C01801=1111.300,173.599,-64.329,-179.246,9.058,149.558
C01802=1111.305,173.385,-64.308,-179.248,9.055,149.558
C01803=1111.309,173.172,-64.289,-179.250,9.053,149.558
C01804=1111.313,172.959,-64.268,-179.252,9.051,149.558
C01805=1111.317,172.746,-64.249,-179.254,9.048,149.558
C01806=1111.321,172.532,-64.228,-179.255,9.045,149.557
C01807=1111.325,172.283,-64.204,-179.258,9.042,149.557
C01808=1111.329,172.035,-64.181,-179.260,9.039,149.557
C01809=1111.334,171.786,-64.158,-179.261,9.037,149.557
C01810=1111.339,171.536,-64.135,-179.264,9.033,149.557
C01811=1111.343,171.288,-64.111,-179.267,9.030,149.557
C01812=1111.348,171.039,-64.087,-179.268,9.028,149.557
C01813=1111.353,170.790,-64.064,-179.271,9.025,149.557
C01814=1111.357,170.541,-64.040,-179.273,9.021,149.557
C01815=1111.362,170.292,-64.017,-179.275,9.018,149.556
C01816=1111.366,170.043,-63.994,-179.277,9.016,149.556
C01817=1111.370,169.795,-63.970,-179.280,9.012,149.556
C01818=1111.375,169.546,-63.947,-179.282,9.009,149.556
C01819=1111.380,169.297,-63.924,-179.284,9.007,149.556
C01820=1111.384,169.048,-63.900,-179.286,9.004,149.556
C01821=1111.389,168.799,-63.877,-179.288,9.000,149.556
C01822=1111.393,168.550,-63.854,-179.290,8.998,149.556
C01823=1111.398,168.301,-63.831,-179.292,8.994,149.555
C01824=1111.403,168.053,-63.808,-179.295,8.991,149.555
C01825=1111.408,167.804,-63.784,-179.297,8.988,149.555
C01826=1111.412,167.555,-63.762,-179.299,8.985,149.555
C01827=1111.416,167.306,-63.738,-179.301,8.982,149.555
C01828=1111.421,167.057,-63.715,-179.304,8.979,149.555
C01829=1111.426,166.808,-63.692,-179.305,8.976,149.555
C01830=1111.430,166.559,-63.669,-179.308,8.973,149.555
C01831=1111.435,166.310,-63.645,-179.310,8.970,149.555
C01832=1111.439,166.061,-63.622,-179.312,8.967,149.555
C01833=1111.445,165.813,-63.599,-179.314,8.964,149.554
C01834=1111.449,165.564,-63.576,-179.316,8.961,149.554
C01835=1111.453,165.315,-63.553,-179.319,8.958,149.554
C01836=1111.458,165.066,-63.530,-179.321,8.954,149.554
C01837=1111.462,164.817,-63.507,-179.323,8.952,149.554
C01838=1111.467,164.568,-63.483,-179.325,8.949,149.554
C01839=1111.472,164.318,-63.461,-179.327,8.945,149.554
C01840=1111.476,164.070,-63.438,-179.330,8.942,149.554
C01841=1111.481,163.821,-63.415,-179.331,8.940,149.553
C01842=1111.486,163.572,-63.392,-179.334,8.936,149.553
C01843=1111.489,163.324,-63.369,-179.336,8.933,149.553
C01844=1111.494,163.075,-63.346,-179.338,8.930,149.553
C01845=1111.498,162.825,-63.324,-179.340,8.927,149.553
C01846=1111.504,162.577,-63.301,-179.342,8.924,149.553
C01847=1111.508,162.328,-63.277,-179.344,8.921,149.553
C01848=1111.512,162.079,-63.254,-179.347,8.917,149.553
C01849=1111.517,161.829,-63.232,-179.349,8.914,149.552
C01850=1111.521,161.581,-63.209,-179.351,8.912,149.552
C01851=1111.527,161.332,-63.186,-179.353,8.908,149.552
C01852=1111.531,161.084,-63.163,-179.356,8.905,149.552
C01853=1111.536,160.834,-63.141,-179.358,8.902,149.552
C01854=1111.540,160.585,-63.117,-179.360,8.898,149.552
C01855=1111.544,160.373,-63.098,-179.362,8.896,149.551
C01856=1111.548,160.159,-63.079,-179.364,8.893,149.551
C01857=1111.552,159.945,-63.059,-179.365,8.891,149.551
C01858=1111.556,159.731,-63.040,-179.368,8.888,149.551
C01859=1111.560,159.518,-63.020,-179.369,8.885,149.551
C01860=1111.564,159.305,-63.000,-179.371,8.883,149.551
C01861=1111.568,159.091,-62.981,-179.373,8.879,149.551
C01862=1111.572,158.877,-62.962,-179.375,8.877,149.551
C01863=1111.576,158.629,-62.939,-179.377,8.873,149.550
C01864=1111.581,158.379,-62.917,-179.379,8.871,149.550
C01865=1111.585,158.131,-62.894,-179.381,8.867,149.550
C01866=1111.590,157.882,-62.871,-179.383,8.864,149.550
C01867=1111.595,157.633,-62.849,-179.385,8.861,149.550
C01868=1111.599,157.384,-62.826,-179.388,8.857,149.550
C01869=1111.604,157.135,-62.804,-179.390,8.854,149.550
C01870=1111.608,156.887,-62.781,-179.392,8.851,149.549
C01871=1111.613,156.637,-62.758,-179.394,8.848,149.549
C01872=1111.617,156.388,-62.736,-179.396,8.845,149.549
C01873=1111.623,156.139,-62.713,-179.398,8.841,149.549
C01874=1111.627,155.891,-62.690,-179.400,8.838,149.549
C01875=1111.631,155.641,-62.668,-179.403,8.835,149.549
C01876=1111.637,155.392,-62.646,-179.405,8.831,149.548
C01877=1111.641,155.144,-62.623,-179.407,8.828,149.548
C01878=1111.645,154.894,-62.601,-179.409,8.824,149.548
C01879=1111.650,154.646,-62.578,-179.412,8.821,149.548
C01880=1111.654,154.397,-62.556,-179.414,8.818,149.548
C01881=1111.659,154.148,-62.535,-179.415,8.815,149.547
C01882=1111.664,153.899,-62.511,-179.417,8.812,149.547
C01883=1111.668,153.650,-62.489,-179.420,8.808,149.547
C01884=1111.673,153.401,-62.467,-179.422,8.805,149.547
C01885=1111.678,153.152,-62.444,-179.424,8.801,149.547
C01886=1111.682,152.902,-62.422,-179.426,8.798,149.546
C01887=1111.687,152.654,-62.400,-179.428,8.794,149.546
C01888=1111.692,152.405,-62.377,-179.430,8.791,149.546
C01889=1111.697,152.156,-62.355,-179.433,8.788,149.546
C01890=1111.701,151.907,-62.333,-179.435,8.784,149.546
C01891=1111.705,151.659,-62.311,-179.437,8.781,149.545
C01892=1111.710,151.409,-62.288,-179.439,8.777,149.545
C01893=1111.715,151.160,-62.266,-179.441,8.774,149.545
C01894=1111.720,150.911,-62.245,-179.443,8.770,149.545
C01895=1111.724,150.662,-62.223,-179.445,8.767,149.544
C01896=1111.729,150.414,-62.200,-179.447,8.763,149.544
C01897=1111.733,150.164,-62.177,-179.449,8.760,149.544
C01898=1111.738,149.916,-62.156,-179.451,8.757,149.544
C01899=1111.743,149.666,-62.134,-179.453,8.753,149.544
C01900=1111.747,149.418,-62.112,-179.456,8.750,149.543
C01901=1111.752,149.168,-62.089,-179.458,8.746,149.543
C01902=1111.757,148.920,-62.067,-179.460,8.743,149.543
C01903=1111.761,148.671,-62.045,-179.462,8.739,149.543
C01904=1111.766,148.422,-62.023,-179.464,8.736,149.542
C01905=1111.770,148.173,-62.001,-179.466,8.732,149.542
C01906=1111.775,147.924,-61.980,-179.468,8.729,149.542
C01907=1111.780,147.675,-61.958,-179.470,8.725,149.542
C01908=1111.785,147.426,-61.935,-179.472,8.722,149.541
C01909=1111.789,147.176,-61.913,-179.474,8.718,149.541
C01910=1111.794,146.928,-61.892,-179.476,8.715,149.541
C01911=1111.798,146.714,-61.873,-179.478,8.711,149.541
C01912=1111.802,146.500,-61.854,-179.480,8.708,149.540
C01913=1111.805,146.287,-61.835,-179.482,8.705,149.540
C01914=1111.810,146.074,-61.816,-179.483,8.702,149.540
C01915=1111.813,145.860,-61.798,-179.485,8.699,149.540
C01916=1111.818,145.646,-61.779,-179.488,8.695,149.540
C01917=1111.822,145.432,-61.760,-179.489,8.692,149.539
C01918=1111.826,145.219,-61.742,-179.491,8.689,149.539
C01919=1111.830,144.970,-61.720,-179.492,8.686,149.539
C01920=1111.835,144.721,-61.698,-179.494,8.682,149.538
C01921=1111.839,144.472,-61.676,-179.496,8.679,149.538
C01922=1111.844,144.223,-61.654,-179.497,8.676,149.538
C01923=1111.849,143.974,-61.632,-179.499,8.672,149.537
C01924=1111.853,143.725,-61.611,-179.501,8.668,149.537
C01925=1111.858,143.476,-61.589,-179.502,8.665,149.537
C01926=1111.863,143.227,-61.567,-179.504,8.662,149.536
C01927=1111.868,142.978,-61.546,-179.506,8.658,149.536
C01928=1111.872,142.728,-61.524,-179.507,8.655,149.536
C01929=1111.877,142.480,-61.502,-179.509,8.652,149.535
C01930=1111.882,142.231,-61.481,-179.511,8.648,149.535
C01931=1111.886,141.982,-61.459,-179.513,8.644,149.535
C01932=1111.891,141.732,-61.438,-179.514,8.641,149.534
C01933=1111.896,141.483,-61.416,-179.516,8.638,149.534
C01934=1111.900,141.235,-61.394,-179.518,8.634,149.534
C01935=1111.905,140.986,-61.373,-179.519,8.631,149.533
C01936=1111.909,140.736,-61.351,-179.521,8.628,149.533
C01937=1111.914,140.488,-61.330,-179.523,8.624,149.533
C01938=1111.919,140.239,-61.308,-179.524,8.621,149.532
C01939=1111.923,139.990,-61.286,-179.526,8.617,149.532
C01940=1111.928,139.740,-61.265,-179.528,8.614,149.532
C01941=1111.933,139.492,-61.243,-179.529,8.611,149.531
C01942=1111.937,139.242,-61.221,-179.531,8.607,149.531
C01943=1111.942,138.993,-61.201,-179.533,8.604,149.531
C01944=1111.947,138.745,-61.179,-179.534,8.601,149.531
C01945=1111.951,138.495,-61.157,-179.536,8.597,149.530
C01946=1111.956,138.246,-61.136,-179.538,8.593,149.530
C01947=1111.961,137.998,-61.115,-179.539,8.591,149.530
C01948=1111.965,137.748,-61.093,-179.541,8.587,149.529
C01949=1111.970,137.499,-61.072,-179.543,8.583,149.529
C01950=1111.975,137.251,-61.051,-179.544,8.581,149.529
C01951=1111.979,137.001,-61.029,-179.546,8.577,149.528
C01952=1111.984,136.752,-61.007,-179.548,8.573,149.528
C01953=1111.989,136.503,-60.987,-179.550,8.571,149.528
C01954=1111.993,136.254,-60.965,-179.551,8.567,149.527
C01955=1111.998,136.004,-60.944,-179.553,8.563,149.527
C01956=1112.003,135.756,-60.922,-179.555,8.560,149.527
C01957=1112.008,135.507,-60.901,-179.556,8.557,149.526
C01958=1112.011,135.258,-60.880,-179.558,8.553,149.526
C01959=1112.017,135.008,-60.859,-179.560,8.550,149.526
C01960=1112.022,134.760,-60.837,-179.562,8.547,149.526
C01961=1112.027,134.510,-60.816,-179.564,8.543,149.525
C01962=1112.031,134.262,-60.795,-179.565,8.540,149.525
C01963=1112.035,134.012,-60.774,-179.567,8.537,149.525
C01964=1112.040,133.763,-60.752,-179.569,8.533,149.524
C01965=1112.045,133.514,-60.732,-179.570,8.530,149.524
C01966=1112.050,133.266,-60.710,-179.572,8.527,149.524
C01967=1112.053,133.051,-60.692,-179.574,8.524,149.524
C01968=1112.058,132.838,-60.674,-179.575,8.521,149.523
C01969=1112.062,132.625,-60.656,-179.576,8.518,149.523
C01970=1112.066,132.410,-60.638,-179.578,8.515,149.523
C01971=1112.069,132.197,-60.620,-179.580,8.512,149.523
C01972=1112.074,131.983,-60.602,-179.581,8.509,149.522
C01973=1112.078,131.769,-60.583,-179.583,8.507,149.522
C01974=1112.082,131.556,-60.565,-179.584,8.504,149.522
C01975=1112.086,131.307,-60.545,-179.586,8.500,149.522
C01976=1112.091,131.058,-60.524,-179.588,8.497,149.521
C01977=1112.096,130.809,-60.502,-179.589,8.494,149.521
C01978=1112.100,130.559,-60.481,-179.591,8.490,149.521
C01979=1112.105,130.310,-60.460,-179.593,8.487,149.521
C01980=1112.110,130.061,-60.440,-179.594,8.484,149.520
C01981=1112.115,129.813,-60.418,-179.596,8.480,149.520
C01982=1112.120,129.563,-60.397,-179.598,8.477,149.520
C01983=1112.124,129.314,-60.377,-179.600,8.474,149.519
C01984=1112.129,129.065,-60.356,-179.601,8.470,149.519
C01985=1112.133,128.816,-60.335,-179.604,8.467,149.519
C01986=1112.138,128.567,-60.314,-179.605,8.464,149.519
C01987=1112.142,128.318,-60.293,-179.607,8.460,149.518
C01988=1112.148,128.069,-60.272,-179.609,8.457,149.518
C01989=1112.153,127.819,-60.251,-179.610,8.454,149.518
C01990=1112.157,127.570,-60.231,-179.612,8.450,149.517
C01991=1112.162,127.322,-60.209,-179.614,8.447,149.517
C01992=1112.167,127.073,-60.189,-179.615,8.444,149.517
C01993=1112.172,126.824,-60.168,-179.617,8.440,149.517
C01994=1112.176,126.574,-60.147,-179.619,8.437,149.516
C01995=1112.180,126.325,-60.127,-179.621,8.434,149.516
C01996=1112.185,126.076,-60.106,-179.622,8.430,149.516
C01997=1112.190,125.827,-60.085,-179.625,8.427,149.515
C01998=1112.195,125.577,-60.064,-179.626,8.424,149.515
C01999=1112.199,125.329,-60.044,-179.628,8.420,149.515
C02000=1112.204,125.080,-60.022,-179.630,8.417,149.515
C02001=1112.209,124.831,-60.002,-179.631,8.414,149.514
C02002=1112.214,124.582,-59.981,-179.633,8.410,149.514
C02003=1112.218,124.333,-59.961,-179.635,8.407,149.514
C02004=1112.223,124.084,-59.940,-179.637,8.403,149.513
C02005=1112.228,123.835,-59.919,-179.638,8.400,149.513
C02006=1112.232,123.586,-59.899,-179.640,8.397,149.513
C02007=1112.237,123.336,-59.878,-179.642,8.393,149.513
C02008=1112.242,123.087,-59.858,-179.644,8.391,149.513
C02009=1112.247,122.838,-59.838,-179.645,8.387,149.512
C02010=1112.252,122.589,-59.817,-179.648,8.383,149.512
C02011=1112.256,122.340,-59.797,-179.649,8.380,149.512
C02012=1112.261,122.091,-59.776,-179.651,8.377,149.511
C02013=1112.266,121.841,-59.755,-179.653,8.373,149.511
C02014=1112.270,121.592,-59.735,-179.654,8.370,149.511
C02015=1112.275,121.343,-59.715,-179.656,8.367,149.511
C02016=1112.280,121.094,-59.694,-179.658,8.363,149.510
C02017=1112.284,120.845,-59.673,-179.660,8.360,149.510
C02018=1112.289,120.596,-59.653,-179.661,8.357,149.510
C02019=1112.294,120.346,-59.633,-179.663,8.353,149.509
C02020=1112.299,120.097,-59.612,-179.665,8.350,149.509
C02021=1112.303,119.849,-59.592,-179.666,8.347,149.509
C02022=1112.307,119.600,-59.571,-179.668,8.343,149.509
C02023=1112.312,119.386,-59.554,-179.670,8.341,149.508
C02024=1112.315,119.171,-59.536,-179.672,8.337,149.508
C02025=1112.320,118.958,-59.519,-179.673,8.334,149.508
C02026=1112.324,118.744,-59.501,-179.675,8.332,149.508
C02027=1112.328,118.530,-59.484,-179.676,8.329,149.507
C02028=1112.332,118.316,-59.467,-179.678,8.326,149.507
C02029=1112.337,118.102,-59.449,-179.679,8.323,149.507
C02030=1112.340,117.890,-59.432,-179.681,8.320,149.507
C02031=1112.345,117.640,-59.411,-179.682,8.317,149.506
C02032=1112.350,117.391,-59.391,-179.684,8.313,149.506
C02033=1112.354,117.142,-59.371,-179.686,8.310,149.506
C02034=1112.359,116.892,-59.351,-179.688,8.306,149.505
C02035=1112.363,116.643,-59.331,-179.689,8.303,149.505
C02036=1112.369,116.394,-59.310,-179.691,8.300,149.505
C02037=1112.373,116.144,-59.290,-179.693,8.296,149.505
C02038=1112.378,115.896,-59.270,-179.695,8.292,149.504
C02039=1112.383,115.647,-59.250,-179.697,8.290,149.504
C02040=1112.388,115.398,-59.230,-179.699,8.286,149.504
C02041=1112.392,115.149,-59.210,-179.700,8.282,149.503
C02042=1112.397,114.899,-59.189,-179.702,8.279,149.503
C02043=1112.402,114.650,-59.169,-179.704,8.276,149.503
C02044=1112.406,114.401,-59.149,-179.705,8.272,149.503
C02045=1112.412,114.152,-59.129,-179.707,8.269,149.502
C02046=1112.416,113.903,-59.109,-179.709,8.265,149.502
C02047=1112.421,113.654,-59.089,-179.710,8.262,149.502
C02048=1112.425,113.405,-59.069,-179.713,8.259,149.501
C02049=1112.430,113.155,-59.049,-179.715,8.255,149.501
C02050=1112.434,112.906,-59.029,-179.716,8.251,149.501
C02051=1112.441,112.657,-59.009,-179.718,8.248,149.501
C02052=1112.445,112.408,-58.989,-179.720,8.245,149.500
C02053=1112.450,112.158,-58.969,-179.721,8.241,149.500
C02054=1112.454,111.909,-58.949,-179.723,8.238,149.500
C02055=1112.459,111.660,-58.929,-179.725,8.235,149.499
C02056=1112.464,111.412,-58.909,-179.726,8.231,149.499
C02057=1112.469,111.162,-58.889,-179.728,8.227,149.499
C02058=1112.473,110.912,-58.870,-179.731,8.224,149.499
C02059=1112.478,110.664,-58.849,-179.733,8.220,149.498
C02060=1112.483,110.414,-58.830,-179.734,8.217,149.498
C02061=1112.488,110.166,-58.810,-179.736,8.213,149.498
C02062=1112.492,109.916,-58.790,-179.738,8.210,149.497
C02063=1112.497,109.667,-58.770,-179.741,8.205,149.497
C02064=1112.502,109.418,-58.750,-179.743,8.202,149.497
C02065=1112.507,109.169,-58.731,-179.745,8.198,149.497
C02066=1112.512,108.919,-58.711,-179.747,8.194,149.496
C02067=1112.516,108.670,-58.691,-179.749,8.191,149.496
C02068=1112.521,108.421,-58.671,-179.750,8.187,149.496
C02069=1112.526,108.172,-58.652,-179.752,8.184,149.495
C02070=1112.530,107.923,-58.632,-179.755,8.180,149.495
C02071=1112.535,107.674,-58.612,-179.756,8.176,149.495
C02072=1112.540,107.425,-58.593,-179.758,8.173,149.495
C02073=1112.545,107.175,-58.573,-179.761,8.168,149.494
C02074=1112.549,106.926,-58.553,-179.762,8.164,149.494
C02075=1112.554,106.677,-58.533,-179.765,8.161,149.494
C02076=1112.559,106.428,-58.514,-179.766,8.157,149.493
C02077=1112.564,106.178,-58.494,-179.768,8.154,149.493
C02078=1112.568,105.929,-58.475,-179.770,8.150,149.493
C02079=1112.572,105.715,-58.458,-179.771,8.147,149.492
C02080=1112.577,105.501,-58.442,-179.773,8.143,149.492
C02081=1112.581,105.288,-58.425,-179.775,8.141,149.492
C02082=1112.585,105.074,-58.408,-179.776,8.137,149.491
C02083=1112.589,104.860,-58.391,-179.778,8.134,149.491
C02084=1112.594,104.646,-58.375,-179.780,8.131,149.491
C02085=1112.597,104.432,-58.358,-179.781,8.128,149.491
C02086=1112.602,104.218,-58.341,-179.783,8.124,149.490
C02087=1112.606,103.969,-58.322,-179.784,8.120,149.490
C02088=1112.611,103.720,-58.302,-179.787,8.117,149.490
C02089=1112.615,103.471,-58.282,-179.788,8.113,149.489
C02090=1112.621,103.222,-58.263,-179.790,8.109,149.489
C02091=1112.625,102.973,-58.244,-179.792,8.105,149.489
C02092=1112.629,102.723,-58.224,-179.793,8.101,149.488
C02093=1112.635,102.474,-58.205,-179.795,8.098,149.488
C02094=1112.640,102.225,-58.185,-179.797,8.094,149.487
C02095=1112.644,101.976,-58.167,-179.799,8.090,149.487
C02096=1112.649,101.726,-58.147,-179.800,8.086,149.487
C02097=1112.654,101.477,-58.127,-179.802,8.083,149.486
C02098=1112.659,101.228,-58.108,-179.804,8.079,149.486
C02099=1112.663,100.978,-58.090,-179.806,8.075,149.486
C02100=1112.669,100.729,-58.070,-179.807,8.071,149.485
C02101=1112.673,100.480,-58.051,-179.809,8.068,149.485
C02102=1112.678,100.231,-58.032,-179.811,8.064,149.484
C02103=1112.683,99.982,-58.012,-179.812,8.060,149.484
C02104=1112.688,99.732,-57.993,-179.814,8.056,149.484
C02105=1112.692,99.483,-57.974,-179.816,8.052,149.483
C02106=1112.697,99.234,-57.954,-179.817,8.048,149.483
C02107=1112.701,98.985,-57.936,-179.819,8.045,149.482
C02108=1112.707,98.735,-57.917,-179.820,8.042,149.482
C02109=1112.712,98.486,-57.897,-179.822,8.038,149.482
C02110=1112.716,98.237,-57.878,-179.823,8.034,149.481
C02111=1112.721,97.988,-57.859,-179.825,8.030,149.481
C02112=1112.726,97.739,-57.839,-179.827,8.026,149.480
C02113=1112.731,97.489,-57.821,-179.828,8.022,149.480
C02114=1112.736,97.240,-57.802,-179.830,8.018,149.479
C02115=1112.740,96.991,-57.783,-179.831,8.014,149.479
C02116=1112.745,96.742,-57.763,-179.833,8.010,149.479
C02117=1112.750,96.493,-57.745,-179.835,8.007,149.478
C02118=1112.755,96.243,-57.726,-179.836,8.003,149.478
C02119=1112.759,95.994,-57.707,-179.838,7.999,149.477
C02120=1112.764,95.745,-57.687,-179.839,7.996,149.477
C02121=1112.769,95.496,-57.670,-179.840,7.992,149.476
C02122=1112.774,95.246,-57.650,-179.842,7.988,149.476
C02123=1112.778,94.998,-57.631,-179.844,7.984,149.476
C02124=1112.783,94.747,-57.612,-179.845,7.980,149.475
C02125=1112.788,94.499,-57.594,-179.847,7.976,149.475
C02126=1112.793,94.250,-57.574,-179.848,7.972,149.474
C02127=1112.798,94.000,-57.556,-179.850,7.969,149.474
C02128=1112.803,93.751,-57.537,-179.851,7.965,149.473
C02129=1112.807,93.501,-57.518,-179.853,7.962,149.473
C02130=1112.813,93.252,-57.499,-179.854,7.958,149.473
C02131=1112.817,93.003,-57.480,-179.855,7.953,149.472
C02132=1112.822,92.754,-57.461,-179.857,7.949,149.471
C02133=1112.827,92.505,-57.443,-179.858,7.946,149.471
C02134=1112.832,92.255,-57.424,-179.859,7.942,149.471
C02135=1112.836,92.042,-57.408,-179.861,7.939,149.470
C02136=1112.840,91.827,-57.392,-179.862,7.935,149.470
C02137=1112.844,91.613,-57.376,-179.863,7.932,149.469
C02138=1112.848,91.399,-57.360,-179.865,7.928,149.469
C02139=1112.853,91.186,-57.343,-179.866,7.926,149.469
C02140=1112.857,90.971,-57.327,-179.867,7.923,149.468
C02141=1112.861,90.757,-57.311,-179.868,7.920,149.468
C02142=1112.865,90.544,-57.295,-179.870,7.916,149.467
C02143=1112.869,90.294,-57.277,-179.871,7.913,149.467
C02144=1112.875,90.045,-57.258,-179.872,7.908,149.466
C02145=1112.879,89.795,-57.239,-179.873,7.904,149.466
C02146=1112.883,89.547,-57.221,-179.875,7.900,149.465
C02147=1112.889,89.297,-57.202,-179.875,7.897,149.465
C02148=1112.893,89.048,-57.183,-179.877,7.893,149.464
C02149=1112.898,88.799,-57.165,-179.879,7.889,149.464
C02150=1112.904,88.549,-57.147,-179.880,7.885,149.463
C02151=1112.908,88.300,-57.127,-179.881,7.882,149.463
C02152=1112.913,88.051,-57.109,-179.882,7.878,149.462
C02153=1112.918,87.802,-57.090,-179.884,7.874,149.462
C02154=1112.922,87.552,-57.072,-179.885,7.870,149.461
C02155=1112.927,87.303,-57.054,-179.886,7.867,149.461
C02156=1112.933,87.054,-57.035,-179.888,7.863,149.460
C02157=1112.937,86.805,-57.017,-179.889,7.858,149.460
C02158=1112.942,86.555,-56.998,-179.890,7.855,149.459
C02159=1112.947,86.306,-56.980,-179.891,7.851,149.459
C02160=1112.952,86.057,-56.961,-179.892,7.847,149.458
C02161=1112.956,85.807,-56.943,-179.893,7.844,149.458
C02162=1112.961,85.558,-56.925,-179.894,7.840,149.457
C02163=1112.966,85.310,-56.906,-179.896,7.836,149.457
C02164=1112.972,85.060,-56.887,-179.897,7.833,149.456
C02165=1112.976,84.810,-56.869,-179.898,7.828,149.456
C02166=1112.981,84.561,-56.851,-179.900,7.825,149.455
C02167=1112.985,84.312,-56.832,-179.900,7.821,149.455
C02168=1112.990,84.063,-56.814,-179.902,7.817,149.454
C02169=1112.995,83.813,-56.795,-179.903,7.813,149.453
C02170=1113.000,83.564,-56.777,-179.904,7.810,149.453
C02171=1113.005,83.315,-56.759,-179.905,7.806,149.452
C02172=1113.010,83.066,-56.741,-179.906,7.802,149.452
C02173=1113.014,82.816,-56.722,-179.908,7.799,149.452
C02174=1113.019,82.567,-56.704,-179.909,7.794,149.451
C02175=1113.025,82.318,-56.686,-179.910,7.791,149.450
C02176=1113.030,82.068,-56.668,-179.911,7.787,149.450
C02177=1113.034,81.819,-56.650,-179.912,7.784,149.449
C02178=1113.039,81.569,-56.632,-179.913,7.779,149.449
C02179=1113.044,81.320,-56.614,-179.914,7.776,149.448
C02180=1113.048,81.072,-56.595,-179.915,7.772,149.448
C02181=1113.053,80.822,-56.577,-179.917,7.768,149.447
C02182=1113.057,80.573,-56.559,-179.917,7.765,149.447
C02183=1113.062,80.323,-56.541,-179.919,7.761,149.446
C02184=1113.068,80.074,-56.522,-179.919,7.757,149.445
C02185=1113.073,79.825,-56.504,-179.920,7.753,149.445
C02186=1113.078,79.576,-56.486,-179.921,7.750,149.444
C02187=1113.083,79.326,-56.468,-179.922,7.746,149.444
C02188=1113.087,79.077,-56.450,-179.923,7.742,149.443
C02189=1113.092,78.827,-56.432,-179.925,7.738,149.443
C02190=1113.097,78.578,-56.414,-179.925,7.735,149.442
C02191=1113.102,78.364,-56.399,-179.926,7.732,149.442
C02192=1113.105,78.150,-56.383,-179.927,7.728,149.441
C02193=1113.110,77.935,-56.367,-179.928,7.725,149.441
C02194=1113.114,77.722,-56.352,-179.929,7.722,149.440
C02195=1113.117,77.508,-56.337,-179.930,7.719,149.440
C02196=1113.122,77.294,-56.321,-179.930,7.716,149.439
C02197=1113.126,77.079,-56.306,-179.931,7.713,149.439
C02198=1113.130,76.866,-56.290,-179.932,7.709,149.438
C02199=1113.135,76.617,-56.272,-179.934,7.706,149.438
C02200=1113.140,76.368,-56.254,-179.935,7.701,149.437
C02201=1113.145,76.117,-56.236,-179.937,7.697,149.437
C02202=1113.150,75.868,-56.218,-179.938,7.693,149.436
C02203=1113.155,75.619,-56.200,-179.940,7.690,149.436
C02204=1113.160,75.370,-56.182,-179.941,7.685,149.435
C02205=1113.164,75.120,-56.164,-179.942,7.682,149.435
C02206=1113.169,74.871,-56.146,-179.943,7.678,149.434
C02207=1113.174,74.622,-56.128,-179.945,7.674,149.434
C02208=1113.179,74.372,-56.111,-179.946,7.670,149.433
C02209=1113.184,74.123,-56.093,-179.948,7.666,149.433
C02210=1113.189,73.874,-56.076,-179.949,7.662,149.433
C02211=1113.193,73.625,-56.058,-179.950,7.658,149.432
C02212=1113.198,73.376,-56.040,-179.952,7.654,149.431
C02213=1113.203,73.125,-56.022,-179.953,7.650,149.431
C02214=1113.208,72.876,-56.004,-179.955,7.646,149.431
C02215=1113.213,72.627,-55.986,-179.956,7.642,149.430
C02216=1113.218,72.378,-55.968,-179.958,7.638,149.429
C02217=1113.223,72.128,-55.951,-179.959,7.635,149.429
C02218=1113.228,71.879,-55.933,-179.960,7.631,149.428
C02219=1113.232,71.630,-55.916,-179.961,7.627,149.428
C02220=1113.237,71.381,-55.898,-179.963,7.623,149.428
C02221=1113.242,71.131,-55.880,-179.965,7.619,149.427
C02222=1113.247,70.882,-55.862,-179.966,7.615,149.426
C02223=1113.252,70.633,-55.844,-179.967,7.611,149.426
C02224=1113.257,70.383,-55.827,-179.969,7.607,149.426
C02225=1113.261,70.134,-55.810,-179.970,7.603,149.425
C02226=1113.266,69.885,-55.792,-179.971,7.599,149.425
C02227=1113.272,69.635,-55.775,-179.973,7.595,149.424
C02228=1113.276,69.386,-55.757,-179.974,7.591,149.423
C02229=1113.281,69.136,-55.740,-179.975,7.587,149.423
C02230=1113.286,68.887,-55.722,-179.977,7.583,149.423
C02231=1113.291,68.638,-55.704,-179.978,7.579,149.422
C02232=1113.296,68.388,-55.687,-179.979,7.575,149.421
C02233=1113.301,68.139,-55.669,-179.981,7.571,149.421
C02234=1113.305,67.890,-55.652,-179.982,7.567,149.420
C02235=1113.311,67.641,-55.634,-179.984,7.563,149.420
C02236=1113.316,67.391,-55.617,-179.985,7.559,149.420
C02237=1113.320,67.143,-55.600,-179.986,7.556,149.419
C02238=1113.325,66.893,-55.583,-179.987,7.552,149.418
C02239=1113.330,66.644,-55.565,-179.988,7.548,149.418
C02240=1113.336,66.394,-55.547,-179.990,7.544,149.417
C02241=1113.340,66.145,-55.530,-179.991,7.540,149.417
C02242=1113.345,65.895,-55.513,-179.993,7.535,149.416
C02243=1113.350,65.646,-55.495,-179.994,7.532,149.416
C02244=1113.354,65.396,-55.478,-179.996,7.528,149.415
C02245=1113.359,65.147,-55.460,-179.997,7.523,149.415
C02246=1113.364,64.898,-55.443,-179.998,7.520,149.414
C02247=1113.369,64.684,-55.428,-179.999,7.516,149.414
C02248=1113.373,64.470,-55.413,180.000,7.513,149.413
C02249=1113.377,64.255,-55.398,179.999,7.510,149.413
C02250=1113.381,64.041,-55.383,179.997,7.506,149.413
C02251=1113.385,63.828,-55.369,179.996,7.503,149.412
C02252=1113.389,63.613,-55.354,179.995,7.500,149.412
C02253=1113.393,63.399,-55.339,179.994,7.496,149.411
C02254=1113.398,63.184,-55.325,179.993,7.493,149.411
C02255=1113.403,62.936,-55.308,179.992,7.489,149.410
C02256=1113.408,62.686,-55.290,179.990,7.485,149.410
C02257=1113.413,62.436,-55.273,179.989,7.480,149.409
C02258=1113.417,62.187,-55.256,179.987,7.477,149.409
C02259=1113.422,61.937,-55.238,179.987,7.473,149.408
C02260=1113.427,61.688,-55.222,179.985,7.469,149.408
C02261=1113.432,61.439,-55.204,179.984,7.465,149.407
C02262=1113.437,61.190,-55.187,179.983,7.461,149.407
C02263=1113.442,60.940,-55.170,179.981,7.457,149.406
C02264=1113.447,60.691,-55.153,179.980,7.453,149.405
C02265=1113.452,60.442,-55.136,179.979,7.449,149.405
C02266=1113.457,60.193,-55.119,179.978,7.445,149.404
C02267=1113.462,59.943,-55.102,179.976,7.441,149.404
C02268=1113.466,59.693,-55.085,179.975,7.437,149.403
C02269=1113.472,59.444,-55.068,179.974,7.433,149.403
C02270=1113.476,59.195,-55.051,179.973,7.429,149.402
C02271=1113.482,58.946,-55.034,179.971,7.425,149.402
C02272=1113.486,58.696,-55.017,179.970,7.421,149.401
C02273=1113.491,58.446,-55.000,179.969,7.418,149.401
C02274=1113.496,58.197,-54.983,179.968,7.414,149.400
C02275=1113.501,57.947,-54.966,179.966,7.409,149.400
C02276=1113.506,57.698,-54.950,179.965,7.405,149.399
C02277=1113.511,57.449,-54.932,179.964,7.401,149.399
C02278=1113.515,57.200,-54.915,179.962,7.397,149.398
C02279=1113.521,56.951,-54.899,179.961,7.393,149.397
C02280=1113.526,56.701,-54.881,179.960,7.390,149.397
C02281=1113.530,56.452,-54.865,179.959,7.386,149.396
C02282=1113.535,56.202,-54.847,179.958,7.382,149.396
C02283=1113.541,55.953,-54.831,179.956,7.377,149.395
C02284=1113.546,55.703,-54.814,179.955,7.373,149.395
C02285=1113.550,55.454,-54.797,179.954,7.369,149.394
C02286=1113.555,55.204,-54.780,179.953,7.366,149.394
C02287=1113.560,54.955,-54.764,179.952,7.362,149.393
C02288=1113.565,54.706,-54.747,179.951,7.357,149.392
C02289=1113.569,54.456,-54.730,179.949,7.354,149.392
C02290=1113.575,54.207,-54.713,179.948,7.349,149.391
C02291=1113.580,53.958,-54.697,179.947,7.345,149.391
C02292=1113.584,53.708,-54.680,179.945,7.341,149.390
C02293=1113.590,53.459,-54.663,179.944,7.338,149.390
C02294=1113.595,53.210,-54.646,179.943,7.334,149.389
C02295=1113.599,52.960,-54.630,179.942,7.329,149.389
C02296=1113.605,52.711,-54.613,179.941,7.325,149.388
C02297=1113.610,52.461,-54.597,179.940,7.321,149.388
C02298=1113.614,52.211,-54.580,179.938,7.317,149.387
C02299=1113.620,51.962,-54.563,179.938,7.314,149.386
C02300=1113.624,51.713,-54.547,179.937,7.309,149.386
C02301=1113.629,51.464,-54.530,179.935,7.305,149.385
C02302=1113.634,51.215,-54.514,179.934,7.301,149.385
C02303=1113.639,51.000,-54.499,179.933,7.298,149.384
C02304=1113.643,50.786,-54.485,179.931,7.294,149.384
C02305=1113.647,50.571,-54.471,179.930,7.291,149.383
C02306=1113.651,50.358,-54.457,179.930,7.287,149.383
C02307=1113.655,50.143,-54.443,179.929,7.284,149.382
C02308=1113.660,49.929,-54.428,179.928,7.280,149.382
C02309=1113.664,49.715,-54.414,179.927,7.277,149.381
C02310=1113.668,49.501,-54.400,179.926,7.274,149.381
C02311=1113.673,49.251,-54.384,179.925,7.270,149.380
C02312=1113.678,49.001,-54.366,179.924,7.266,149.380
C02313=1113.683,48.752,-54.351,179.922,7.261,149.379
C02314=1113.688,48.502,-54.334,179.921,7.257,149.379
C02315=1113.693,48.254,-54.318,179.920,7.253,149.378
C02316=1113.697,48.004,-54.301,179.919,7.250,149.377
C02317=1113.702,47.754,-54.285,179.918,7.246,149.377
C02318=1113.707,47.505,-54.269,179.917,7.241,149.376
C02319=1113.712,47.255,-54.252,179.916,7.237,149.376
C02320=1113.718,47.006,-54.236,179.914,7.233,149.375
C02321=1113.722,46.757,-54.219,179.913,7.229,149.375
C02322=1113.727,46.508,-54.203,179.913,7.225,149.374
C02323=1113.732,46.258,-54.187,179.911,7.221,149.373
C02324=1113.737,46.009,-54.171,179.910,7.217,149.373
C02325=1113.742,45.759,-54.154,179.909,7.213,149.372
C02326=1113.747,45.510,-54.139,179.908,7.208,149.371
C02327=1113.752,45.260,-54.122,179.907,7.204,149.371
C02328=1113.757,45.010,-54.105,179.906,7.201,149.370
C02329=1113.762,44.761,-54.089,179.905,7.197,149.370
C02330=1113.767,44.512,-54.072,179.904,7.192,149.369
C02331=1113.772,44.262,-54.057,179.902,7.189,149.369
C02332=1113.777,44.013,-54.040,179.901,7.184,149.368
C02333=1113.782,43.764,-54.025,179.900,7.180,149.367
C02334=1113.786,43.514,-54.008,179.899,7.176,149.367
C02335=1113.792,43.265,-53.992,179.898,7.172,149.366
C02336=1113.797,43.016,-53.976,179.897,7.168,149.366
C02337=1113.802,42.766,-53.960,179.896,7.164,149.365
C02338=1113.807,42.517,-53.944,179.895,7.160,149.364
C02339=1113.812,42.267,-53.928,179.894,7.156,149.364
C02340=1113.817,42.018,-53.911,179.893,7.152,149.363
C02341=1113.821,41.768,-53.896,179.892,7.148,149.363
C02342=1113.827,41.519,-53.879,179.890,7.144,149.362
C02343=1113.831,41.269,-53.863,179.889,7.139,149.361
C02344=1113.837,41.020,-53.848,179.888,7.135,149.361
C02345=1113.841,40.770,-53.831,179.888,7.131,149.360
C02346=1113.847,40.521,-53.815,179.887,7.127,149.359
C02347=1113.852,40.272,-53.799,179.885,7.123,149.359
C02348=1113.856,40.022,-53.783,179.884,7.119,149.358
C02349=1113.862,39.773,-53.768,179.883,7.115,149.358
C02350=1113.866,39.523,-53.751,179.882,7.110,149.357
C02351=1113.871,39.274,-53.736,179.882,7.107,149.356
C02352=1113.875,39.024,-53.719,179.881,7.102,149.356
C02353=1113.881,38.775,-53.704,179.879,7.098,149.355
C02354=1113.886,38.526,-53.688,179.878,7.094,149.355
C02355=1113.891,38.276,-53.671,179.877,7.090,149.354
C02356=1113.896,38.027,-53.656,179.876,7.086,149.353
C02357=1113.901,37.777,-53.640,179.875,7.082,149.353
C02358=1113.906,37.527,-53.624,179.874,7.078,149.352
C02359=1113.911,37.313,-53.611,179.873,7.073,149.351
C02360=1113.915,37.099,-53.597,179.872,7.070,149.351
C02361=1113.919,36.884,-53.583,179.872,7.067,149.350
C02362=1113.923,36.670,-53.570,179.871,7.064,149.350
C02363=1113.927,36.456,-53.556,179.870,7.059,149.349
C02364=1113.931,36.242,-53.543,179.869,7.056,149.349
C02365=1113.936,36.027,-53.529,179.868,7.053,149.348
C02366=1113.940,35.813,-53.515,179.867,7.049,149.348
C02367=1113.945,35.564,-53.500,179.866,7.045,149.347
C02368=1113.951,35.314,-53.484,179.865,7.041,149.346
C02369=1113.955,35.064,-53.468,179.864,7.037,149.346
C02370=1113.960,34.815,-53.453,179.863,7.032,149.345
C02371=1113.965,34.566,-53.437,179.862,7.028,149.344
C02372=1113.970,34.316,-53.421,179.861,7.024,149.344
C02373=1113.975,34.067,-53.405,179.861,7.020,149.343
C02374=1113.981,33.817,-53.390,179.860,7.016,149.342
C02375=1113.985,33.568,-53.375,179.859,7.012,149.342
C02376=1113.990,33.318,-53.359,179.858,7.007,149.341
C02377=1113.996,33.069,-53.343,179.856,7.003,149.340
C02378=1114.001,32.819,-53.328,179.855,6.999,149.340
C02379=1114.005,32.570,-53.311,179.855,6.995,149.339
C02380=1114.010,32.321,-53.296,179.854,6.990,149.338
C02381=1114.015,32.071,-53.280,179.853,6.986,149.338
C02382=1114.020,31.822,-53.265,179.852,6.982,149.337
C02383=1114.025,31.572,-53.249,179.851,6.978,149.336
C02384=1114.030,31.323,-53.234,179.850,6.973,149.336
C02385=1114.036,31.073,-53.218,179.849,6.969,149.335
C02386=1114.040,30.824,-53.203,179.849,6.965,149.334
C02387=1114.045,30.574,-53.187,179.848,6.961,149.334
C02388=1114.050,30.325,-53.172,179.846,6.957,149.333
C02389=1114.055,30.076,-53.157,179.845,6.952,149.332
C02390=1114.061,29.826,-53.141,179.845,6.948,149.331
C02391=1114.065,29.576,-53.125,179.844,6.943,149.331
C02392=1114.070,29.327,-53.110,179.843,6.940,149.330
C02393=1114.075,29.078,-53.095,179.842,6.936,149.329
C02394=1114.080,28.829,-53.080,179.841,6.931,149.329
C02395=1114.085,28.578,-53.064,179.840,6.927,149.328
C02396=1114.090,28.329,-53.048,179.839,6.923,149.328
C02397=1114.095,28.080,-53.033,179.839,6.918,149.327
C02398=1114.100,27.830,-53.018,179.838,6.914,149.326
C02399=1114.105,27.581,-53.003,179.837,6.910,149.325
C02400=1114.110,27.331,-52.987,179.836,6.906,149.325
C02401=1114.115,27.081,-52.972,179.835,6.902,149.324
C02402=1114.120,26.832,-52.957,179.834,6.897,149.323
C02403=1114.125,26.583,-52.941,179.833,6.893,149.322
C02404=1114.130,26.334,-52.926,179.832,6.888,149.322
C02405=1114.135,26.084,-52.910,179.832,6.885,149.321
C02406=1114.140,25.834,-52.896,179.831,6.880,149.320
C02407=1114.145,25.584,-52.880,179.830,6.876,149.320
C02408=1114.151,25.335,-52.865,179.829,6.871,149.319
C02409=1114.155,25.086,-52.850,179.828,6.867,149.318
C02410=1114.161,24.837,-52.834,179.828,6.862,149.317
C02411=1114.166,24.587,-52.820,179.826,6.858,149.317
C02412=1114.170,24.337,-52.804,179.826,6.855,149.316
C02413=1114.175,24.088,-52.789,179.825,6.850,149.315
C02414=1114.180,23.838,-52.773,179.824,6.845,149.315
C02415=1114.184,23.624,-52.761,179.824,6.842,149.314
C02416=1114.189,23.409,-52.748,179.823,6.838,149.313
C02417=1114.194,23.195,-52.734,179.822,6.834,149.313
C02418=1114.198,22.980,-52.722,179.822,6.831,149.312
C02419=1114.202,22.766,-52.708,179.821,6.827,149.312
C02420=1114.206,22.551,-52.696,179.820,6.823,149.311
C02421=1114.211,22.337,-52.683,179.820,6.820,149.310
C02422=1114.215,22.123,-52.670,179.819,6.815,149.310
C02423=1114.220,21.874,-52.655,179.818,6.811,149.309
C02424=1114.225,21.624,-52.640,179.818,6.807,149.308
C02425=1114.230,21.375,-52.625,179.817,6.803,149.307
C02426=1114.235,21.124,-52.610,179.816,6.798,149.307
C02427=1114.240,20.875,-52.595,179.815,6.794,149.306
C02428=1114.245,20.626,-52.580,179.814,6.789,149.305
C02429=1114.250,20.376,-52.565,179.813,6.785,149.304
C02430=1114.255,20.127,-52.550,179.812,6.780,149.304
C02431=1114.260,19.878,-52.535,179.812,6.776,149.303
C02432=1114.265,19.628,-52.520,179.811,6.772,149.302
C02433=1114.270,19.378,-52.505,179.811,6.767,149.301
C02434=1114.275,19.129,-52.491,179.810,6.763,149.301
C02435=1114.280,18.879,-52.475,179.809,6.759,149.300
C02436=1114.285,18.630,-52.461,179.808,6.754,149.299
C02437=1114.290,18.381,-52.446,179.807,6.750,149.298
C02438=1114.296,18.131,-52.431,179.807,6.745,149.298
C02439=1114.300,17.881,-52.416,179.805,6.741,149.297
C02440=1114.305,17.632,-52.402,179.806,6.737,149.296
C02441=1114.311,17.382,-52.386,179.805,6.732,149.295
C02442=1114.316,17.133,-52.372,179.804,6.728,149.294
C02443=1114.320,16.884,-52.357,179.803,6.723,149.294
C02444=1114.326,16.634,-52.342,179.802,6.719,149.293
C02445=1114.330,16.384,-52.327,179.802,6.714,149.292
C02446=1114.335,16.135,-52.313,179.801,6.710,149.291
C02447=1114.341,15.885,-52.297,179.800,6.705,149.290
C02448=1114.346,15.636,-52.283,179.799,6.701,149.290
C02449=1114.350,15.387,-52.268,179.799,6.697,149.289
C02450=1114.355,15.137,-52.253,179.799,6.692,149.288
C02451=1114.361,14.887,-52.239,179.798,6.688,149.287
C02452=1114.366,14.638,-52.224,179.797,6.683,149.287
C02453=1114.371,14.388,-52.209,179.796,6.678,149.286
C02454=1114.375,14.139,-52.194,179.795,6.674,149.285
C02455=1114.381,13.889,-52.179,179.795,6.669,149.284
C02456=1114.386,13.639,-52.165,179.794,6.665,149.283
C02457=1114.391,13.390,-52.150,179.793,6.660,149.283
C02458=1114.396,13.140,-52.136,179.793,6.656,149.282
C02459=1114.401,12.891,-52.122,179.793,6.652,149.281
C02460=1114.406,12.641,-52.106,179.792,6.647,149.280
C02461=1114.411,12.392,-52.092,179.791,6.643,149.279
C02462=1114.416,12.143,-52.078,179.791,6.638,149.278
C02463=1114.421,11.893,-52.064,179.790,6.634,149.278
C02464=1114.426,11.644,-52.049,179.789,6.629,149.277
C02465=1114.431,11.394,-52.034,179.789,6.624,149.276
C02466=1114.437,11.144,-52.019,179.788,6.620,149.275
C02467=1114.441,10.895,-52.004,179.787,6.615,149.274
C02468=1114.446,10.645,-51.990,179.786,6.610,149.274
C02469=1114.451,10.395,-51.976,179.786,6.606,149.273
C02470=1114.456,10.146,-51.962,179.786,6.602,149.272
C02471=1114.461,9.932,-51.950,179.785,6.598,149.271
C02472=1114.465,9.717,-51.937,179.784,6.594,149.270
C02473=1114.470,9.503,-51.925,179.784,6.589,149.270
C02474=1114.474,9.288,-51.912,179.784,6.586,149.269
C02475=1114.478,9.073,-51.899,179.783,6.582,149.268
C02476=1114.483,8.859,-51.887,179.782,6.578,149.268
C02477=1114.487,8.645,-51.875,179.782,6.574,149.267
C02478=1114.491,8.430,-51.862,179.782,6.570,149.266
C02479=1114.497,8.181,-51.848,179.781,6.566,149.265
C02480=1114.502,7.931,-51.834,179.781,6.561,149.264
C02481=1114.507,7.681,-51.819,179.780,6.556,149.263
C02482=1114.512,7.432,-51.805,179.779,6.552,149.263
C02483=1114.517,7.182,-51.791,179.779,6.547,149.262
C02484=1114.521,6.932,-51.776,179.778,6.543,149.261
C02485=1114.527,6.683,-51.763,179.777,6.538,149.260
C02486=1114.532,6.434,-51.748,179.777,6.533,149.259
C02487=1114.537,6.184,-51.733,179.776,6.528,149.258
C02488=1114.542,5.935,-51.719,179.775,6.524,149.258
C02489=1114.547,5.685,-51.705,179.775,6.520,149.257
C02490=1114.552,5.436,-51.691,179.775,6.515,149.256
C02491=1114.557,5.186,-51.676,179.774,6.511,149.255
C02492=1114.562,4.937,-51.662,179.774,6.506,149.254
C02493=1114.567,4.687,-51.648,179.773,6.502,149.253
C02494=1114.572,4.437,-51.634,179.772,6.497,149.253
C02495=1114.577,4.188,-51.620,179.772,6.492,149.252
C02496=1114.582,3.938,-51.605,179.771,6.488,149.251
C02497=1114.587,3.689,-51.591,179.771,6.483,149.250
C02498=1114.592,3.439,-51.577,179.770,6.479,149.249
C02499=1114.598,3.190,-51.563,179.770,6.475,149.248
C02500=1114.603,2.940,-51.549,179.769,6.470,149.247
C02501=1114.608,2.691,-51.534,179.769,6.465,149.247
C02502=1114.613,2.440,-51.521,179.768,6.461,149.246
C02503=1114.619,2.191,-51.507,179.767,6.456,149.245
C02504=1114.623,1.942,-51.493,179.767,6.451,149.244
C02505=1114.628,1.692,-51.479,179.766,6.447,149.243
C02506=1114.633,1.442,-51.465,179.765,6.442,149.243
C02507=1114.638,1.193,-51.451,179.764,6.438,149.242
C02508=1114.643,0.944,-51.437,179.765,6.434,149.241
C02509=1114.648,0.694,-51.422,179.764,6.429,149.240
C02510=1114.654,0.445,-51.408,179.763,6.425,149.239
C02511=1114.659,0.195,-51.395,179.763,6.420,149.238
C02512=1114.663,-0.055,-51.381,179.762,6.415,149.237
C02513=1114.668,-0.304,-51.367,179.761,6.411,149.237
C02514=1114.674,-0.553,-51.353,179.760,6.406,149.236
C02515=1114.679,-0.803,-51.339,179.760,6.401,149.235
C02516=1114.684,-1.053,-51.325,179.759,6.397,149.234
C02517=1114.690,-1.302,-51.311,179.759,6.393,149.233
C02518=1114.694,-1.552,-51.298,179.758,6.389,149.233
C02519=1114.699,-1.802,-51.283,179.758,6.384,149.232
C02520=1114.704,-2.051,-51.269,179.757,6.379,149.231
C02521=1114.710,-2.301,-51.256,179.756,6.375,149.230
C02522=1114.714,-2.551,-51.241,179.756,6.370,149.229
C02523=1114.720,-2.800,-51.228,179.755,6.365,149.228
C02524=1114.724,-3.049,-51.214,179.754,6.361,149.228
C02525=1114.729,-3.299,-51.200,179.754,6.356,149.227
C02526=1114.735,-3.548,-51.186,179.754,6.352,149.226
C02527=1114.739,-3.764,-51.175,179.753,6.348,149.225
C02528=1114.744,-3.978,-51.163,179.753,6.344,149.225
C02529=1114.748,-4.193,-51.151,179.752,6.340,149.224
C02530=1114.752,-4.407,-51.139,179.752,6.336,149.223
C02531=1114.756,-4.622,-51.127,179.751,6.333,149.222
C02532=1114.761,-4.836,-51.115,179.750,6.328,149.222
C02533=1114.766,-5.051,-51.104,179.750,6.325,149.221
C02534=1114.770,-5.266,-51.092,179.750,6.321,149.220
C02535=1114.775,-5.515,-51.078,179.749,6.317,149.220
C02536=1114.780,-5.764,-51.065,179.748,6.312,149.219
C02537=1114.785,-6.015,-51.051,179.747,6.307,149.218
C02538=1114.790,-6.264,-51.037,179.747,6.303,149.217
C02539=1114.795,-6.513,-51.023,179.746,6.298,149.216
C02540=1114.801,-6.763,-51.010,179.745,6.294,149.216
C02541=1114.806,-7.012,-50.996,179.745,6.289,149.215
C02542=1114.811,-7.263,-50.982,179.745,6.285,149.214
C02543=1114.816,-7.511,-50.969,179.745,6.280,149.213
C02544=1114.821,-7.762,-50.956,179.744,6.276,149.212
C02545=1114.826,-8.011,-50.942,179.743,6.271,149.211
C02546=1114.831,-8.261,-50.929,179.743,6.267,149.210
C02547=1114.836,-8.510,-50.915,179.742,6.262,149.210
C02548=1114.841,-8.760,-50.902,179.741,6.257,149.209
C02549=1114.847,-9.009,-50.888,179.741,6.253,149.208
C02550=1114.852,-9.259,-50.874,179.740,6.248,149.207
C02551=1114.856,-9.508,-50.861,179.739,6.244,149.206
C02552=1114.862,-9.758,-50.848,179.738,6.239,149.205
C02553=1114.866,-10.007,-50.834,179.738,6.234,149.205
C02554=1114.872,-10.257,-50.821,179.738,6.231,149.204
C02555=1114.878,-10.563,-50.804,179.737,6.225,149.203
C02556=1114.884,-10.869,-50.788,179.736,6.219,149.202
C02557=1114.891,-11.175,-50.771,179.735,6.213,149.201
C02558=1114.898,-11.480,-50.755,179.735,6.207,149.200
C02559=1114.902,-11.729,-50.741,179.734,6.203,149.199
C02560=1114.908,-11.979,-50.728,179.733,6.198,149.198
C02561=1114.912,-12.228,-50.714,179.733,6.194,149.197
C02562=1114.918,-12.478,-50.701,179.733,6.190,149.196
C02563=1114.922,-12.728,-50.688,179.732,6.185,149.196
C02564=1114.928,-12.977,-50.674,179.731,6.181,149.195
C02565=1114.932,-13.227,-50.661,179.731,6.176,149.194
C02566=1114.938,-13.476,-50.648,179.730,6.171,149.193
C02567=1114.942,-13.726,-50.634,179.729,6.167,149.192
C02568=1114.948,-13.975,-50.621,179.729,6.162,149.191
C02569=1114.953,-14.225,-50.608,179.728,6.157,149.191
C02570=1114.958,-14.474,-50.594,179.728,6.153,149.190
C02571=1114.963,-14.724,-50.582,179.727,6.148,149.189
C02572=1114.969,-14.974,-50.568,179.726,6.144,149.188
C02573=1114.974,-15.223,-50.556,179.726,6.139,149.187
C02574=1114.978,-15.473,-50.542,179.725,6.134,149.186
C02575=1114.984,-15.722,-50.529,179.725,6.129,149.185
C02576=1114.988,-15.972,-50.516,179.724,6.125,149.185
C02577=1114.994,-16.222,-50.503,179.723,6.120,149.184
C02578=1114.999,-16.471,-50.489,179.723,6.116,149.183
C02579=1115.004,-16.721,-50.476,179.722,6.111,149.182
C02580=1115.009,-16.970,-50.463,179.722,6.106,149.181
C02581=1115.014,-17.220,-50.450,179.721,6.101,149.180
C02582=1115.020,-17.470,-50.437,179.720,6.097,149.180
C02583=1115.027,-17.843,-50.417,179.720,6.090,149.178
C02584=1115.035,-18.217,-50.398,179.719,6.083,149.177
C02585=1115.042,-18.590,-50.379,179.718,6.076,149.176
C02586=1115.050,-18.963,-50.359,179.717,6.069,149.174
C02587=1115.056,-19.212,-50.346,179.716,6.064,149.174
C02588=1115.060,-19.462,-50.333,179.716,6.060,149.173
C02589=1115.065,-19.712,-50.320,179.716,6.055,149.172
C02590=1115.071,-19.962,-50.306,179.715,6.050,149.171
C02591=1115.076,-20.211,-50.294,179.715,6.045,149.170
C02592=1115.081,-20.461,-50.281,179.714,6.041,149.169
C02593=1115.086,-20.711,-50.268,179.714,6.036,149.168
C02594=1115.091,-20.960,-50.255,179.713,6.032,149.167
C02595=1115.096,-21.210,-50.243,179.712,6.027,149.167
C02596=1115.102,-21.459,-50.229,179.712,6.022,149.166
C02597=1115.107,-21.709,-50.216,179.711,6.017,149.165
C02598=1115.112,-21.959,-50.204,179.711,6.013,149.164
C02599=1115.117,-22.208,-50.191,179.710,6.008,149.163
C02600=1115.122,-22.458,-50.178,179.710,6.003,149.162
C02601=1115.128,-22.708,-50.165,179.709,5.999,149.161
C02602=1115.133,-22.957,-50.152,179.709,5.994,149.160
C02603=1115.138,-23.206,-50.140,179.708,5.989,149.159
C02604=1115.143,-23.457,-50.126,179.708,5.984,149.159
C02605=1115.148,-23.706,-50.114,179.707,5.980,149.158
C02606=1115.153,-23.955,-50.101,179.707,5.975,149.157
C02607=1115.158,-24.205,-50.088,179.706,5.970,149.156
C02608=1115.164,-24.455,-50.075,179.706,5.965,149.155
C02609=1115.169,-24.704,-50.062,179.705,5.960,149.154
C02610=1115.174,-24.953,-50.050,179.704,5.955,149.153
C02611=1115.179,-25.204,-50.037,179.704,5.950,149.152
C02612=1115.184,-25.453,-50.025,179.703,5.946,149.151
C02613=1115.190,-25.703,-50.012,179.703,5.941,149.150
C02614=1115.195,-25.952,-49.999,179.704,5.937,149.149
C02615=1115.200,-26.202,-49.986,179.703,5.932,149.148
C02616=1115.204,-26.452,-49.973,179.704,5.928,149.147
C02617=1115.210,-26.702,-49.962,179.704,5.923,149.146
C02618=1115.215,-26.951,-49.949,179.704,5.919,149.145
C02619=1115.220,-27.200,-49.936,179.705,5.915,149.144
C02620=1115.225,-27.451,-49.923,179.705,5.911,149.143
C02621=1115.231,-27.700,-49.910,179.706,5.907,149.142
C02622=1115.236,-27.949,-49.898,179.705,5.902,149.141
C02623=1115.241,-28.199,-49.886,179.706,5.898,149.140
C02624=1115.246,-28.448,-49.873,179.706,5.894,149.139
C02625=1115.251,-28.699,-49.860,179.706,5.890,149.138
C02626=1115.256,-28.948,-49.848,179.706,5.885,149.137
C02627=1115.261,-29.198,-49.836,179.706,5.881,149.136
C02628=1115.266,-29.447,-49.823,179.707,5.877,149.135
C02629=1115.272,-29.696,-49.810,179.706,5.872,149.134
C02630=1115.277,-29.947,-49.797,179.707,5.868,149.133
C02631=1115.282,-30.197,-49.785,179.707,5.864,149.132
C02632=1115.287,-30.446,-49.772,179.706,5.859,149.131
C02633=1115.292,-30.695,-49.760,179.707,5.855,149.130
C02634=1115.298,-30.945,-49.747,179.706,5.850,149.130
C02635=1115.302,-31.159,-49.737,179.706,5.846,149.129
C02636=1115.306,-31.375,-49.726,179.706,5.843,149.128
C02637=1115.310,-31.590,-49.716,179.706,5.839,149.127
C02638=1115.315,-31.804,-49.704,179.706,5.835,149.126
C02639=1115.320,-32.019,-49.694,179.705,5.832,149.126
C02640=1115.324,-32.234,-49.683,179.705,5.828,149.125
C02641=1115.329,-32.448,-49.673,179.705,5.824,149.124
C02642=1115.333,-32.663,-49.662,179.705,5.820,149.123
C02643=1115.338,-32.914,-49.649,179.704,5.816,149.123
C02644=1115.343,-33.163,-49.637,179.704,5.812,149.122
C02645=1115.349,-33.412,-49.624,179.704,5.807,149.121
C02646=1115.354,-33.662,-49.612,179.704,5.803,149.120
C02647=1115.359,-33.912,-49.600,179.703,5.798,149.119
C02648=1115.364,-34.161,-49.587,179.703,5.794,149.118
C02649=1115.370,-34.411,-49.575,179.703,5.789,149.117
C02650=1115.375,-34.660,-49.563,179.702,5.785,149.116
C02651=1115.380,-34.911,-49.550,179.701,5.780,149.116
C02652=1115.385,-35.160,-49.538,179.701,5.775,149.115
C02653=1115.389,-35.410,-49.526,179.701,5.771,149.114
C02654=1115.395,-35.659,-49.514,179.700,5.766,149.113
C02655=1115.400,-35.909,-49.502,179.699,5.762,149.112
C02656=1115.405,-36.158,-49.489,179.699,5.757,149.111
C02657=1115.410,-36.408,-49.477,179.698,5.752,149.110
C02658=1115.416,-36.658,-49.465,179.697,5.748,149.110
C02659=1115.421,-36.907,-49.452,179.697,5.743,149.109
C02660=1115.426,-37.157,-49.440,179.696,5.738,149.108
C02661=1115.431,-37.406,-49.428,179.695,5.734,149.107
C02662=1115.437,-37.656,-49.416,179.695,5.729,149.106
C02663=1115.442,-37.906,-49.404,179.694,5.724,149.105
C02664=1115.447,-38.155,-49.391,179.694,5.719,149.104
C02665=1115.452,-38.405,-49.380,179.693,5.715,149.104
C02666=1115.456,-38.655,-49.367,179.692,5.710,149.103
C02667=1115.462,-38.905,-49.355,179.691,5.704,149.102
C02668=1115.467,-39.154,-49.343,179.690,5.700,149.101
C02669=1115.472,-39.404,-49.331,179.689,5.694,149.100
C02670=1115.478,-39.654,-49.319,179.689,5.690,149.100
C02671=1115.483,-39.903,-49.306,179.687,5.684,149.099
C02672=1115.488,-40.153,-49.295,179.687,5.680,149.098
C02673=1115.493,-40.403,-49.283,179.686,5.674,149.097
C02674=1115.498,-40.652,-49.270,179.685,5.669,149.096
C02675=1115.504,-40.902,-49.259,179.684,5.664,149.095
C02676=1115.510,-41.151,-49.247,179.683,5.660,149.095
C02677=1115.514,-41.400,-49.235,179.682,5.654,149.094
C02678=1115.520,-41.650,-49.223,179.681,5.648,149.093
C02679=1115.525,-41.900,-49.211,179.680,5.643,149.092
C02680=1115.530,-42.150,-49.199,179.679,5.638,149.091
C02681=1115.536,-42.400,-49.187,179.678,5.633,149.090
C02682=1115.540,-42.649,-49.176,179.677,5.627,149.089
C02683=1115.546,-42.899,-49.164,179.676,5.622,149.088
C02684=1115.551,-43.148,-49.151,179.676,5.617,149.088
C02685=1115.555,-43.398,-49.140,179.676,5.612,149.086
C02686=1115.561,-43.648,-49.128,179.676,5.608,149.085
C02687=1115.566,-43.898,-49.116,179.676,5.603,149.084
C02688=1115.572,-44.148,-49.104,179.677,5.599,149.083
C02689=1115.576,-44.397,-49.092,179.677,5.593,149.082
C02690=1115.582,-44.647,-49.080,179.677,5.588,149.081
C02691=1115.586,-44.862,-49.070,179.677,5.584,149.080
C02692=1115.590,-45.077,-49.060,179.677,5.580,149.079
C02693=1115.595,-45.291,-49.050,179.677,5.577,149.078
C02694=1115.600,-45.507,-49.040,179.677,5.573,149.077
C02695=1115.605,-45.721,-49.030,179.678,5.569,149.076
C02696=1115.609,-45.936,-49.020,179.678,5.565,149.075
C02697=1115.613,-46.150,-49.010,179.678,5.561,149.074
C02698=1115.618,-46.365,-49.000,179.678,5.557,149.074
C02699=1115.623,-46.615,-48.988,179.678,5.552,149.072
C02700=1115.628,-46.865,-48.976,179.678,5.547,149.071
C02701=1115.633,-47.115,-48.965,179.678,5.543,149.070
C02702=1115.639,-47.365,-48.953,179.678,5.537,149.069
C02703=1115.643,-47.614,-48.941,179.679,5.533,149.068
C02704=1115.648,-47.864,-48.929,179.679,5.528,149.067
C02705=1115.654,-48.113,-48.918,179.679,5.523,149.066
C02706=1115.659,-48.363,-48.906,179.679,5.519,149.065
C02707=1115.665,-48.613,-48.894,179.680,5.514,149.064
C02708=1115.670,-48.862,-48.883,179.679,5.509,149.063
C02709=1115.675,-49.112,-48.871,179.680,5.505,149.062
C02710=1115.680,-49.362,-48.859,179.680,5.500,149.061
C02711=1115.685,-49.611,-48.848,179.680,5.496,149.060
C02712=1115.691,-49.861,-48.837,179.680,5.490,149.058
C02713=1115.696,-50.111,-48.825,179.680,5.485,149.057
C02714=1115.701,-50.360,-48.813,179.680,5.481,149.056
C02715=1115.706,-50.610,-48.801,179.680,5.476,149.055
C02716=1115.711,-50.860,-48.790,179.681,5.472,149.054
C02717=1115.717,-51.109,-48.779,179.681,5.467,149.053
C02718=1115.722,-51.359,-48.767,179.681,5.462,149.052
C02719=1115.727,-51.609,-48.755,179.681,5.458,149.051
C02720=1115.732,-51.858,-48.744,179.682,5.453,149.050
C02721=1115.737,-52.108,-48.732,179.682,5.449,149.049
C02722=1115.743,-52.357,-48.721,179.682,5.443,149.048
C02723=1115.748,-52.607,-48.709,179.682,5.438,149.047
C02724=1115.753,-52.857,-48.698,179.682,5.434,149.046
C02725=1115.758,-53.107,-48.686,179.682,5.429,149.044
C02726=1115.763,-53.357,-48.676,179.683,5.425,149.043
C02727=1115.769,-53.606,-48.664,179.682,5.420,149.042
C02728=1115.774,-53.856,-48.653,179.683,5.415,149.041
C02729=1115.779,-54.106,-48.641,179.683,5.411,149.040
C02730=1115.784,-54.355,-48.630,179.683,5.406,149.039
C02731=1115.789,-54.605,-48.618,179.684,5.402,149.038
C02732=1115.795,-54.854,-48.607,179.684,5.396,149.037
C02733=1115.800,-55.104,-48.595,179.683,5.392,149.036
C02734=1115.805,-55.354,-48.584,179.684,5.387,149.035
C02735=1115.811,-55.604,-48.573,179.684,5.382,149.034
C02736=1115.816,-55.853,-48.562,179.684,5.378,149.033
C02737=1115.821,-56.103,-48.550,179.684,5.373,149.032
C02738=1115.826,-56.353,-48.539,179.684,5.368,149.031
C02739=1115.831,-56.603,-48.527,179.685,5.364,149.029
C02740=1115.837,-56.852,-48.516,179.685,5.359,149.028
C02741=1115.842,-57.102,-48.505,179.684,5.354,149.027
C02742=1115.847,-57.352,-48.493,179.685,5.350,149.026
C02743=1115.852,-57.602,-48.482,179.685,5.345,149.025
C02744=1115.857,-57.851,-48.471,179.685,5.341,149.024
C02745=1115.863,-58.101,-48.460,179.685,5.336,149.023
C02746=1115.868,-58.351,-48.449,179.685,5.331,149.022
C02747=1115.872,-58.566,-48.439,179.685,5.327,149.021
C02748=1115.877,-58.780,-48.429,179.685,5.323,149.020
C02749=1115.882,-58.995,-48.420,179.686,5.319,149.019
C02750=1115.886,-59.210,-48.410,179.686,5.315,149.018
C02751=1115.890,-59.425,-48.400,179.686,5.311,149.017
C02752=1115.895,-59.640,-48.390,179.686,5.307,149.017
C02753=1115.899,-59.855,-48.380,179.686,5.303,149.016
C02754=1115.904,-60.070,-48.371,179.687,5.299,149.015
C02755=1115.909,-60.320,-48.360,179.686,5.294,149.014
C02756=1115.914,-60.569,-48.349,179.685,5.289,149.013
C02757=1115.920,-60.819,-48.337,179.684,5.283,149.012
C02758=1115.925,-61.069,-48.327,179.684,5.278,149.011
C02759=1115.930,-61.318,-48.315,179.684,5.274,149.010
C02760=1115.935,-61.567,-48.305,179.683,5.268,149.009
C02761=1115.941,-61.818,-48.293,179.683,5.263,149.008
C02762=1115.945,-62.068,-48.282,179.682,5.258,149.007
C02763=1115.951,-62.317,-48.272,179.681,5.253,149.006
C02764=1115.956,-62.567,-48.260,179.681,5.248,149.005
C02765=1115.961,-62.817,-48.249,179.680,5.242,149.004
C02766=1115.967,-63.066,-48.238,179.680,5.237,149.003
C02767=1115.971,-63.316,-48.227,179.679,5.233,149.002
C02768=1115.977,-63.566,-48.216,179.679,5.227,149.001
C02769=1115.982,-63.815,-48.205,179.679,5.222,149.000
C02770=1115.987,-64.066,-48.195,179.678,5.216,148.999
C02771=1115.993,-64.314,-48.184,179.677,5.212,148.998
C02772=1115.998,-64.564,-48.172,179.677,5.206,148.997
C02773=1116.003,-64.815,-48.161,179.676,5.201,148.996
C02774=1116.008,-65.064,-48.150,179.677,5.196,148.995
C02775=1116.013,-65.314,-48.140,179.676,5.191,148.994
C02776=1116.019,-65.563,-48.129,179.675,5.185,148.993
C02777=1116.024,-65.813,-48.118,179.675,5.180,148.992
C02778=1116.030,-66.062,-48.107,179.675,5.176,148.991
C02779=1116.035,-66.312,-48.096,179.674,5.170,148.990
C02780=1116.040,-66.563,-48.085,179.674,5.165,148.989
C02781=1116.045,-66.812,-48.075,179.674,5.160,148.988
C02782=1116.050,-67.062,-48.064,179.674,5.155,148.987
C02783=1116.056,-67.311,-48.052,179.673,5.149,148.986
C02784=1116.061,-67.561,-48.042,179.673,5.144,148.985
C02785=1116.066,-67.810,-48.031,179.673,5.139,148.984
C02786=1116.071,-68.061,-48.020,179.672,5.134,148.983
C02787=1116.077,-68.310,-48.010,179.672,5.128,148.982
C02788=1116.082,-68.560,-47.999,179.672,5.124,148.981
C02789=1116.087,-68.809,-47.989,179.672,5.118,148.980
C02790=1116.092,-69.059,-47.978,179.672,5.113,148.978
C02791=1116.098,-69.309,-47.967,179.671,5.108,148.978
C02792=1116.103,-69.559,-47.956,179.671,5.103,148.976
C02793=1116.109,-69.809,-47.946,179.671,5.098,148.975
C02794=1116.113,-70.058,-47.934,179.670,5.092,148.974
C02795=1116.119,-70.308,-47.924,179.671,5.087,148.973
C02796=1116.124,-70.558,-47.914,179.670,5.082,148.972
C02797=1116.129,-70.807,-47.903,179.670,5.077,148.971
C02798=1116.134,-71.057,-47.892,179.670,5.071,148.970
C02799=1116.140,-71.307,-47.882,179.670,5.066,148.969
C02800=1116.145,-71.557,-47.871,179.670,5.061,148.968
C02801=1116.150,-71.806,-47.861,179.670,5.056,148.967
C02802=1116.155,-72.056,-47.850,179.670,5.051,148.965
C02803=1116.160,-72.271,-47.841,179.670,5.046,148.965
C02804=1116.165,-72.486,-47.832,179.669,5.041,148.964
C02805=1116.169,-72.701,-47.823,179.669,5.037,148.963
C02806=1116.174,-72.916,-47.814,179.669,5.032,148.962
C02807=1116.178,-73.131,-47.805,179.669,5.029,148.961
C02808=1116.182,-73.346,-47.795,179.669,5.024,148.960
C02809=1116.188,-73.561,-47.786,179.669,5.019,148.959
C02810=1116.192,-73.776,-47.778,179.669,5.015,148.958
C02811=1116.197,-74.026,-47.768,179.670,5.009,148.957
C02812=1116.202,-74.276,-47.757,179.669,5.004,148.956
C02813=1116.208,-74.525,-47.746,179.669,4.999,148.955
C02814=1116.213,-74.775,-47.736,179.669,4.994,148.953
C02815=1116.218,-75.025,-47.725,179.669,4.988,148.952
C02816=1116.224,-75.274,-47.715,179.669,4.983,148.951
C02817=1116.229,-75.525,-47.705,179.669,4.978,148.950
C02818=1116.234,-75.774,-47.694,179.669,4.973,148.949
C02819=1116.240,-76.024,-47.684,179.670,4.968,148.947
C02820=1116.245,-76.274,-47.674,179.670,4.963,148.946
C02821=1116.251,-76.523,-47.663,179.669,4.958,148.945
C02822=1116.256,-76.773,-47.653,179.669,4.952,148.944
C02823=1116.261,-77.023,-47.643,179.669,4.947,148.943
C02824=1116.266,-77.272,-47.632,179.669,4.942,148.942
C02825=1116.271,-77.522,-47.622,179.669,4.937,148.941
C02826=1116.276,-77.772,-47.611,179.670,4.931,148.940
C02827=1116.282,-78.021,-47.601,179.670,4.926,148.938
C02828=1116.287,-78.271,-47.591,179.670,4.921,148.937
C02829=1116.292,-78.521,-47.580,179.670,4.916,148.936
C02830=1116.298,-78.770,-47.570,179.670,4.911,148.935
C02831=1116.303,-79.021,-47.560,179.670,4.906,148.934
C02832=1116.309,-79.270,-47.549,179.671,4.900,148.933
C02833=1116.313,-79.520,-47.540,179.671,4.895,148.931
C02834=1116.319,-79.769,-47.530,179.671,4.890,148.930
C02835=1116.324,-80.019,-47.519,179.671,4.885,148.929
C02836=1116.330,-80.269,-47.510,179.671,4.880,148.928
C02837=1116.336,-80.519,-47.499,179.671,4.875,148.927
C02838=1116.340,-80.769,-47.489,179.671,4.870,148.925
C02839=1116.345,-81.018,-47.479,179.672,4.864,148.924
C02840=1116.351,-81.268,-47.469,179.672,4.859,148.923
C02841=1116.356,-81.518,-47.458,179.672,4.854,148.922
C02842=1116.362,-81.768,-47.448,179.673,4.849,148.921
C02843=1116.367,-82.017,-47.439,179.673,4.844,148.919
C02844=1116.372,-82.267,-47.428,179.674,4.839,148.918
C02845=1116.377,-82.517,-47.418,179.674,4.834,148.917
C02846=1116.383,-82.766,-47.408,179.674,4.829,148.916
C02847=1116.388,-83.016,-47.399,179.674,4.824,148.915
C02848=1116.393,-83.266,-47.388,179.674,4.818,148.914
C02849=1116.398,-83.516,-47.378,179.674,4.813,148.912
C02850=1116.404,-83.766,-47.368,179.675,4.808,148.911
C02851=1116.409,-84.015,-47.358,179.675,4.804,148.910
C02852=1116.414,-84.265,-47.347,179.676,4.798,148.909
C02853=1116.420,-84.515,-47.338,179.676,4.793,148.907
C02854=1116.425,-84.765,-47.328,179.676,4.788,148.906
C02855=1116.430,-85.014,-47.318,179.677,4.783,148.905
C02856=1116.435,-85.264,-47.308,179.677,4.778,148.904
C02857=1116.441,-85.514,-47.297,179.678,4.773,148.903
C02858=1116.446,-85.764,-47.288,179.678,4.768,148.902
C02859=1116.451,-85.979,-47.279,179.678,4.764,148.900
C02860=1116.455,-86.194,-47.271,179.678,4.759,148.899
C02861=1116.460,-86.409,-47.262,179.679,4.755,148.898
C02862=1116.465,-86.624,-47.254,179.679,4.751,148.897
C02863=1116.469,-86.839,-47.245,179.680,4.746,148.896
C02864=1116.474,-87.054,-47.236,179.680,4.742,148.895
C02865=1116.478,-87.270,-47.228,179.680,4.738,148.894
C02866=1116.483,-87.484,-47.220,179.681,4.733,148.893
C02867=1116.488,-87.734,-47.210,179.681,4.728,148.892
C02868=1116.493,-87.984,-47.199,179.682,4.724,148.891
C02869=1116.498,-88.234,-47.190,179.682,4.719,148.889
C02870=1116.504,-88.484,-47.180,179.682,4.714,148.888
C02871=1116.509,-88.733,-47.170,179.683,4.709,148.887
C02872=1116.515,-88.983,-47.161,179.683,4.704,148.886
C02873=1116.520,-89.233,-47.151,179.684,4.698,148.884
C02874=1116.525,-89.482,-47.141,179.684,4.694,148.883
C02875=1116.530,-89.733,-47.131,179.685,4.689,148.882
C02876=1116.536,-89.982,-47.121,179.685,4.684,148.881
C02877=1116.541,-90.231,-47.112,179.686,4.679,148.880
C02878=1116.547,-90.482,-47.102,179.686,4.674,148.878
C02879=1116.551,-90.731,-47.092,179.687,4.670,148.877
C02880=1116.557,-90.981,-47.082,179.687,4.664,148.876
C02881=1116.562,-91.231,-47.073,179.688,4.660,148.875
C02882=1116.567,-91.480,-47.063,179.689,4.655,148.873
C02883=1116.573,-91.730,-47.053,179.689,4.649,148.872
C02884=1116.578,-91.980,-47.044,179.690,4.645,148.871
C02885=1116.584,-92.229,-47.033,179.690,4.640,148.870
C02886=1116.588,-92.480,-47.024,179.691,4.636,148.869
C02887=1116.594,-92.729,-47.014,179.691,4.630,148.867
C02888=1116.599,-92.979,-47.005,179.692,4.626,148.866
C02889=1116.605,-93.229,-46.995,179.692,4.620,148.865
C02890=1116.610,-93.478,-46.985,179.693,4.616,148.864
C02891=1116.615,-93.728,-46.976,179.693,4.611,148.862
C02892=1116.621,-93.978,-46.966,179.694,4.607,148.861
C02893=1116.626,-94.228,-46.957,179.695,4.602,148.860
C02894=1116.631,-94.478,-46.946,179.695,4.597,148.859
C02895=1116.636,-94.728,-46.937,179.695,4.592,148.858
C02896=1116.642,-94.977,-46.927,179.696,4.588,148.857
C02897=1116.647,-95.227,-46.918,179.696,4.582,148.855
C02898=1116.653,-95.477,-46.908,179.697,4.577,148.854
C02899=1116.658,-95.727,-46.899,179.697,4.572,148.853
C02900=1116.664,-95.976,-46.889,179.698,4.568,148.852
C02901=1116.669,-96.226,-46.880,179.698,4.563,148.851
C02902=1116.674,-96.475,-46.870,179.698,4.557,148.849
C02903=1116.679,-96.725,-46.861,179.698,4.552,148.848
C02904=1116.685,-96.975,-46.851,179.699,4.548,148.847
C02905=1116.690,-97.225,-46.842,179.699,4.543,148.846
C02906=1116.694,-97.475,-46.832,179.699,4.538,148.845
C02907=1116.700,-97.725,-46.822,179.700,4.532,148.843
C02908=1116.706,-97.975,-46.813,179.700,4.528,148.842
C02909=1116.711,-98.224,-46.803,179.701,4.523,148.841
C02910=1116.716,-98.474,-46.794,179.701,4.518,148.840
C02911=1116.722,-98.724,-46.784,179.701,4.513,148.839
C02912=1116.727,-98.973,-46.775,179.701,4.508,148.838
C02913=1116.732,-99.223,-46.765,179.702,4.504,148.837
C02914=1116.738,-99.473,-46.756,179.702,4.498,148.835
C02915=1116.743,-99.688,-46.748,179.703,4.494,148.834
C02916=1116.747,-99.903,-46.740,179.702,4.489,148.833
C02917=1116.751,-100.118,-46.732,179.703,4.485,148.832
C02918=1116.757,-100.334,-46.724,179.703,4.481,148.831
C02919=1116.761,-100.549,-46.715,179.704,4.477,148.830
C02920=1116.766,-100.764,-46.707,179.703,4.472,148.829
C02921=1116.770,-100.980,-46.700,179.704,4.468,148.828
C02922=1116.774,-101.194,-46.691,179.705,4.464,148.827
C02923=1116.780,-101.444,-46.682,179.704,4.459,148.826
C02924=1116.785,-101.694,-46.673,179.704,4.454,148.825
C02925=1116.790,-101.943,-46.663,179.705,4.449,148.824
C02926=1116.796,-102.194,-46.654,179.706,4.444,148.822
C02927=1116.801,-102.443,-46.645,179.706,4.439,148.821
C02928=1116.807,-102.693,-46.636,179.706,4.434,148.820
C02929=1116.812,-102.943,-46.626,179.706,4.429,148.819
C02930=1116.817,-103.193,-46.617,179.706,4.424,148.818
C02931=1116.822,-103.443,-46.608,179.707,4.419,148.816
C02932=1116.828,-103.692,-46.598,179.707,4.414,148.815
C02933=1116.833,-103.942,-46.589,179.708,4.409,148.814
C02934=1116.838,-104.192,-46.580,179.708,4.404,148.813
C02935=1116.844,-104.442,-46.571,179.708,4.399,148.812
C02936=1116.849,-104.691,-46.561,179.708,4.394,148.810
C02937=1116.854,-104.941,-46.552,179.709,4.388,148.809
C02938=1116.860,-105.191,-46.543,179.709,4.383,148.808
C02939=1116.865,-105.441,-46.533,179.710,4.379,148.807
C02940=1116.871,-105.691,-46.525,179.710,4.374,148.806
C02941=1116.875,-105.940,-46.515,179.710,4.369,148.805
C02942=1116.881,-106.189,-46.506,179.710,4.363,148.803
C02943=1116.887,-106.439,-46.497,179.711,4.358,148.802
C02944=1116.892,-106.689,-46.488,179.711,4.353,148.801
C02945=1116.897,-106.939,-46.479,179.711,4.348,148.800
C02946=1116.903,-107.189,-46.470,179.711,4.343,148.799
C02947=1116.909,-107.439,-46.461,179.712,4.338,148.797
C02948=1116.913,-107.688,-46.451,179.712,4.333,148.796
C02949=1116.919,-107.938,-46.442,179.713,4.328,148.795
C02950=1116.924,-108.188,-46.433,179.713,4.323,148.794
C02951=1116.929,-108.438,-46.424,179.713,4.318,148.793
C02952=1116.935,-108.688,-46.415,179.713,4.313,148.791
C02953=1116.941,-108.937,-46.406,179.714,4.307,148.790
C02954=1116.946,-109.187,-46.398,179.714,4.302,148.789
C02955=1116.951,-109.437,-46.389,179.714,4.297,148.788
C02956=1116.956,-109.687,-46.380,179.714,4.292,148.787
C02957=1116.962,-109.937,-46.370,179.715,4.287,148.785
C02958=1116.967,-110.186,-46.361,179.716,4.282,148.784
C02959=1116.972,-110.436,-46.352,179.716,4.277,148.783
C02960=1116.977,-110.686,-46.343,179.716,4.272,148.782
C02961=1116.983,-110.935,-46.334,179.716,4.267,148.781
C02962=1116.988,-111.185,-46.325,179.717,4.262,148.779
C02963=1116.993,-111.435,-46.316,179.717,4.257,148.778
C02964=1116.999,-111.685,-46.307,179.717,4.251,148.777
C02965=1117.004,-111.935,-46.298,179.717,4.246,148.776
C02966=1117.009,-112.185,-46.289,179.718,4.241,148.775
C02967=1117.015,-112.434,-46.280,179.718,4.236,148.773
C02968=1117.020,-112.684,-46.272,179.718,4.231,148.772
C02969=1117.026,-112.933,-46.263,179.718,4.226,148.771
C02970=1117.031,-113.183,-46.254,179.719,4.220,148.770
C02971=1117.036,-113.399,-46.247,179.719,4.216,148.768
C02972=1117.040,-113.615,-46.239,179.719,4.211,148.768
C02973=1117.045,-113.830,-46.231,179.719,4.207,148.767
C02974=1117.050,-114.045,-46.224,179.720,4.202,148.765
C02975=1117.055,-114.260,-46.216,179.720,4.198,148.764
C02976=1117.059,-114.475,-46.209,179.720,4.193,148.763
C02977=1117.064,-114.691,-46.201,179.721,4.189,148.762
C02978=1117.068,-114.906,-46.193,179.720,4.184,148.761
C02979=1117.074,-115.156,-46.184,179.721,4.179,148.760
C02980=1117.079,-115.406,-46.175,179.721,4.174,148.759
C02981=1117.084,-115.655,-46.167,179.722,4.168,148.757
C02982=1117.090,-115.905,-46.159,179.722,4.163,148.756
C02983=1117.095,-116.155,-46.150,179.722,4.158,148.755
C02984=1117.100,-116.405,-46.141,179.723,4.153,148.754
C02985=1117.106,-116.654,-46.132,179.723,4.148,148.753
C02986=1117.111,-116.904,-46.123,179.723,4.143,148.751
C02987=1117.116,-117.154,-46.114,179.723,4.137,148.750
C02988=1117.122,-117.404,-46.106,179.724,4.132,148.749
C02989=1117.128,-117.654,-46.098,179.724,4.127,148.748
C02990=1117.133,-117.903,-46.089,179.724,4.122,148.747
C02991=1117.138,-118.153,-46.080,179.725,4.116,148.745
C02992=1117.143,-118.403,-46.071,179.725,4.111,148.744
C02993=1117.149,-118.653,-46.063,179.726,4.106,148.743
C02994=1117.154,-118.903,-46.054,179.725,4.100,148.741
C02995=1117.160,-119.153,-46.045,179.725,4.095,148.740
C02996=1117.165,-119.402,-46.037,179.726,4.090,148.739
C02997=1117.170,-119.652,-46.028,179.726,4.084,148.738
C02998=1117.176,-119.902,-46.020,179.727,4.079,148.736
C02999=1117.181,-120.152,-46.011,179.727,4.074,148.735
C03000=1117.187,-120.401,-46.002,179.727,4.069,148.734
C03001=1117.192,-120.651,-45.995,179.728,4.063,148.733
C03002=1117.197,-120.901,-45.986,179.728,4.058,148.732
C03003=1117.203,-121.150,-45.977,179.728,4.052,148.730
C03004=1117.208,-121.401,-45.969,179.728,4.047,148.729
C03005=1117.213,-121.651,-45.960,179.729,4.042,148.728
C03006=1117.219,-121.900,-45.952,179.729,4.036,148.726
C03007=1117.224,-122.150,-45.943,179.729,4.031,148.725
C03008=1117.230,-122.400,-45.935,179.730,4.026,148.724
C03009=1117.235,-122.650,-45.926,179.730,4.020,148.723
C03010=1117.241,-122.900,-45.918,179.730,4.014,148.721
C03011=1117.245,-123.149,-45.910,179.730,4.009,148.720
C03012=1117.251,-123.398,-45.901,179.731,4.004,148.719
C03013=1117.256,-123.649,-45.893,179.732,3.999,148.717
C03014=1117.262,-123.899,-45.884,179.732,3.993,148.716
C03015=1117.268,-124.148,-45.876,179.732,3.987,148.715
C03016=1117.273,-124.398,-45.867,179.732,3.982,148.714
C03017=1117.277,-124.648,-45.859,179.733,3.977,148.712
C03018=1117.283,-124.898,-45.851,179.733,3.972,148.711
C03019=1117.289,-125.147,-45.842,179.733,3.966,148.710
C03020=1117.294,-125.398,-45.834,179.733,3.960,148.709
C03021=1117.300,-125.647,-45.826,179.734,3.955,148.707
C03022=1117.305,-125.897,-45.818,179.734,3.950,148.706
C03023=1117.310,-126.146,-45.809,179.734,3.944,148.705
C03024=1117.316,-126.397,-45.801,179.735,3.938,148.703
C03025=1117.321,-126.647,-45.792,179.735,3.933,148.702
C03026=1117.327,-126.896,-45.785,179.735,3.928,148.701
C03027=1117.331,-127.111,-45.778,179.736,3.923,148.700
C03028=1117.336,-127.327,-45.771,179.735,3.918,148.699
C03029=1117.341,-127.542,-45.763,179.736,3.913,148.697
C03030=1117.344,-127.758,-45.756,179.736,3.909,148.697
C03031=1117.350,-127.973,-45.749,179.736,3.903,148.695
C03032=1117.355,-128.189,-45.742,179.737,3.899,148.694
C03033=1117.359,-128.404,-45.735,179.737,3.894,148.693
C03034=1117.364,-128.619,-45.728,179.737,3.889,148.692
C03035=1116.941,-128.610,-45.754,179.745,3.894,148.691
C03036=1116.936,-128.394,-45.760,179.745,3.899,148.692
C03037=1116.931,-128.179,-45.768,179.744,3.903,148.693
C03038=1116.927,-127.964,-45.775,179.744,3.908,148.694
C03039=1116.922,-127.748,-45.782,179.744,3.913,148.695
C03040=1116.917,-127.533,-45.790,179.743,3.917,148.696
C03041=1116.913,-127.318,-45.796,179.743,3.922,148.697
C03042=1116.908,-127.103,-45.803,179.743,3.927,148.698
C03043=1116.903,-126.886,-45.811,179.742,3.931,148.699
C03044=1116.898,-126.637,-45.819,179.742,3.938,148.701
C03045=1116.893,-126.387,-45.827,179.742,3.943,148.702
C03046=1116.887,-126.138,-45.835,179.742,3.948,148.703
C03047=1116.882,-125.887,-45.844,179.741,3.953,148.705
C03048=1116.876,-125.638,-45.852,179.741,3.959,148.706
C03049=1116.871,-125.389,-45.860,179.741,3.965,148.707
C03050=1116.866,-125.138,-45.869,179.740,3.970,148.709
C03051=1116.861,-124.888,-45.878,179.740,3.975,148.710
C03052=1116.855,-124.639,-45.885,179.739,3.980,148.711
C03053=1116.849,-124.389,-45.894,179.740,3.986,148.712
C03054=1116.844,-124.138,-45.902,179.739,3.992,148.714
C03055=1116.839,-123.889,-45.910,179.738,3.997,148.715
C03056=1116.834,-123.640,-45.919,179.738,4.002,148.716
C03057=1116.828,-123.390,-45.927,179.738,4.008,148.717
C03058=1116.823,-123.140,-45.936,179.738,4.014,148.719
C03059=1116.817,-122.890,-45.945,179.737,4.019,148.720
C03060=1116.812,-122.640,-45.953,179.737,4.024,148.721
C03061=1116.806,-122.390,-45.962,179.737,4.029,148.723
C03062=1116.801,-122.141,-45.970,179.737,4.035,148.724
C03063=1116.796,-121.890,-45.979,179.736,4.040,148.725
C03064=1116.790,-121.641,-45.987,179.736,4.046,148.726
C03065=1116.785,-121.391,-45.995,179.736,4.051,148.728
C03066=1116.780,-121.142,-46.004,179.735,4.056,148.729
C03067=1116.774,-120.892,-46.012,179.735,4.062,148.730
C03068=1116.769,-120.642,-46.021,179.734,4.067,148.731
C03069=1116.764,-120.392,-46.030,179.734,4.072,148.733
C03070=1116.758,-120.142,-46.038,179.734,4.078,148.734
C03071=1116.753,-119.893,-46.047,179.733,4.083,148.735
C03072=1116.747,-119.643,-46.056,179.734,4.089,148.736
C03073=1116.742,-119.393,-46.064,179.734,4.094,148.738
C03074=1116.736,-119.144,-46.073,179.733,4.099,148.739
C03075=1116.731,-118.893,-46.081,179.732,4.105,148.740
C03076=1116.726,-118.643,-46.090,179.732,4.110,148.741
C03077=1116.721,-118.393,-46.099,179.732,4.115,148.743
C03078=1116.715,-118.144,-46.108,179.732,4.120,148.744
C03079=1116.710,-117.895,-46.116,179.731,4.125,148.745
C03080=1116.704,-117.644,-46.125,179.731,4.130,148.746
C03081=1116.699,-117.394,-46.134,179.730,4.136,148.748
C03082=1116.693,-117.145,-46.142,179.730,4.141,148.749
C03083=1116.688,-116.895,-46.151,179.730,4.146,148.750
C03084=1116.683,-116.645,-46.160,179.729,4.151,148.751
C03085=1116.678,-116.395,-46.169,179.729,4.157,148.753
C03086=1116.673,-116.146,-46.178,179.729,4.162,148.754
C03087=1116.667,-115.896,-46.185,179.729,4.168,148.755
C03088=1116.661,-115.646,-46.194,179.729,4.173,148.756
C03089=1116.656,-115.396,-46.203,179.729,4.178,148.757
C03090=1116.651,-115.146,-46.212,179.728,4.184,148.759
C03091=1116.646,-114.896,-46.221,179.728,4.189,148.760
C03092=1116.641,-114.681,-46.229,179.727,4.193,148.761
C03093=1116.636,-114.466,-46.236,179.728,4.198,148.762
C03094=1116.631,-114.251,-46.244,179.727,4.202,148.763
C03095=1116.627,-114.036,-46.252,179.726,4.206,148.764
C03096=1116.622,-113.820,-46.259,179.726,4.211,148.765
C03097=1116.618,-113.605,-46.267,179.726,4.215,148.766
C03098=1116.613,-113.390,-46.275,179.726,4.220,148.767
C03099=1116.608,-113.175,-46.282,179.725,4.224,148.768
C03100=1116.603,-112.925,-46.291,179.725,4.229,148.770
C03101=1116.598,-112.675,-46.300,179.725,4.235,148.771
C03102=1116.592,-112.425,-46.309,179.724,4.240,148.772
C03103=1116.587,-112.176,-46.318,179.724,4.245,148.773
C03104=1116.582,-111.926,-46.327,179.724,4.250,148.774
C03105=1116.576,-111.676,-46.336,179.724,4.255,148.776
C03106=1116.570,-111.426,-46.345,179.723,4.260,148.777
C03107=1116.565,-111.177,-46.354,179.723,4.266,148.778
C03108=1116.560,-110.927,-46.363,179.723,4.271,148.779
C03109=1116.555,-110.677,-46.372,179.723,4.276,148.780
C03110=1116.550,-110.427,-46.380,179.722,4.281,148.782
C03111=1116.544,-110.177,-46.390,179.722,4.286,148.783
C03112=1116.539,-109.927,-46.399,179.722,4.291,148.784
C03113=1116.533,-109.678,-46.407,179.722,4.297,148.785
C03114=1116.528,-109.428,-46.416,179.721,4.301,148.786
C03115=1116.523,-109.178,-46.425,179.721,4.306,148.788
C03116=1116.517,-108.929,-46.435,179.720,4.311,148.789
C03117=1116.512,-108.679,-46.444,179.720,4.316,148.790
C03118=1116.507,-108.429,-46.453,179.720,4.322,148.791
C03119=1116.502,-108.179,-46.462,179.720,4.327,148.792
C03120=1116.496,-107.929,-46.472,179.719,4.332,148.794
C03121=1116.490,-107.679,-46.480,179.719,4.337,148.795
C03122=1116.485,-107.429,-46.489,179.719,4.342,148.796
C03123=1116.480,-107.180,-46.499,179.719,4.347,148.797
C03124=1116.475,-106.930,-46.508,179.718,4.352,148.798
C03125=1116.469,-106.681,-46.517,179.718,4.357,148.800
C03126=1116.464,-106.431,-46.526,179.717,4.362,148.801
C03127=1116.458,-106.181,-46.535,179.717,4.367,148.802
C03128=1116.453,-105.931,-46.545,179.717,4.372,148.803
C03129=1116.448,-105.682,-46.554,179.717,4.378,148.804
C03130=1116.442,-105.432,-46.563,179.716,4.383,148.806
C03131=1116.437,-105.182,-46.572,179.716,4.388,148.807
C03132=1116.431,-104.932,-46.581,179.715,4.392,148.808
C03133=1116.427,-104.682,-46.591,179.715,4.397,148.809
C03134=1116.421,-104.433,-46.600,179.715,4.403,148.810
C03135=1116.415,-104.182,-46.609,179.715,4.408,148.812
C03136=1116.410,-103.933,-46.618,179.714,4.413,148.813
C03137=1116.405,-103.683,-46.628,179.714,4.418,148.814
C03138=1116.400,-103.433,-46.637,179.713,4.422,148.815
C03139=1116.394,-103.183,-46.646,179.713,4.428,148.816
C03140=1116.390,-102.934,-46.656,179.713,4.433,148.818
C03141=1116.384,-102.684,-46.665,179.713,4.438,148.819
C03142=1116.378,-102.434,-46.674,179.712,4.443,148.820
C03143=1116.374,-102.185,-46.684,179.712,4.448,148.821
C03144=1116.368,-101.935,-46.693,179.711,4.453,148.822
C03145=1116.363,-101.685,-46.702,179.711,4.458,148.824
C03146=1116.358,-101.436,-46.712,179.711,4.463,148.825
C03147=1116.352,-101.185,-46.721,179.711,4.468,148.826
C03148=1116.348,-100.970,-46.729,179.710,4.472,148.827
C03149=1116.343,-100.755,-46.738,179.710,4.476,148.828
C03150=1116.338,-100.540,-46.745,179.710,4.481,148.829
C03151=1116.334,-100.324,-46.753,179.710,4.485,148.830
C03152=1116.329,-100.110,-46.762,179.709,4.489,148.831
C03153=1116.324,-99.894,-46.770,179.709,4.493,148.832
C03154=1116.320,-99.679,-46.778,179.709,4.498,148.833
C03155=1116.315,-99.464,-46.786,179.708,4.502,148.834
C03156=1116.309,-99.214,-46.795,179.708,4.507,148.835
C03157=1116.304,-98.965,-46.805,179.707,4.512,148.836
C03158=1116.299,-98.715,-46.814,179.707,4.517,148.838
C03159=1116.294,-98.465,-46.824,179.707,4.522,148.839
C03160=1116.289,-98.216,-46.833,179.707,4.527,148.840
C03161=1116.283,-97.966,-46.843,179.707,4.532,148.841
C03162=1116.278,-97.715,-46.853,179.706,4.536,148.842
C03163=1116.272,-97.465,-46.862,179.706,4.541,148.843
C03164=1116.268,-97.216,-46.872,179.706,4.547,148.845
C03165=1116.262,-96.966,-46.881,179.706,4.552,148.846
C03166=1116.257,-96.717,-46.891,179.705,4.556,148.847
C03167=1116.251,-96.466,-46.900,179.705,4.561,148.848
C03168=1116.246,-96.217,-46.910,179.704,4.566,148.849
C03169=1116.240,-95.967,-46.919,179.704,4.572,148.851
C03170=1116.235,-95.718,-46.929,179.703,4.576,148.852
C03171=1116.229,-95.468,-46.938,179.703,4.581,148.853
C03172=1116.225,-95.218,-46.948,179.703,4.586,148.854
C03173=1116.219,-94.968,-46.958,179.702,4.591,148.855
C03174=1116.214,-94.718,-46.968,179.702,4.596,148.856
C03175=1116.209,-94.469,-46.978,179.702,4.601,148.858
C03176=1116.204,-94.219,-46.987,179.701,4.605,148.859
C03177=1116.198,-93.969,-46.997,179.701,4.610,148.860
C03178=1116.193,-93.720,-47.006,179.700,4.615,148.861
C03179=1116.187,-93.470,-47.016,179.700,4.620,148.862
C03180=1116.182,-93.220,-47.025,179.699,4.624,148.864
C03181=1116.177,-92.970,-47.035,179.698,4.630,148.865
C03182=1116.171,-92.720,-47.046,179.698,4.634,148.866
C03183=1116.166,-92.471,-47.055,179.697,4.639,148.867
C03184=1116.161,-92.221,-47.065,179.697,4.644,148.869
C03185=1116.156,-91.971,-47.074,179.696,4.649,148.870
C03186=1116.150,-91.722,-47.084,179.696,4.653,148.871
C03187=1116.145,-91.472,-47.093,179.695,4.659,148.872
C03188=1116.140,-91.221,-47.103,179.695,4.664,148.874
C03189=1116.134,-90.972,-47.114,179.694,4.668,148.875
C03190=1116.129,-90.723,-47.123,179.694,4.673,148.876
C03191=1116.123,-90.473,-47.133,179.693,4.678,148.877
C03192=1116.119,-90.223,-47.142,179.693,4.683,148.878
C03193=1116.113,-89.974,-47.152,179.692,4.688,148.880
C03194=1116.108,-89.723,-47.162,179.691,4.693,148.881
C03195=1116.103,-89.474,-47.172,179.691,4.698,148.882
C03196=1116.097,-89.224,-47.182,179.690,4.702,148.883
C03197=1116.091,-88.974,-47.192,179.690,4.707,148.884
C03198=1116.086,-88.725,-47.201,179.690,4.713,148.886
C03199=1116.081,-88.474,-47.212,179.689,4.717,148.887
C03200=1116.076,-88.225,-47.222,179.688,4.722,148.888
C03201=1116.071,-87.975,-47.231,179.688,4.728,148.889
C03202=1116.065,-87.726,-47.241,179.687,4.732,148.891
C03203=1116.060,-87.475,-47.252,179.687,4.737,148.892
C03204=1116.056,-87.261,-47.260,179.687,4.741,148.893
C03205=1116.051,-87.045,-47.268,179.687,4.746,148.894
C03206=1116.046,-86.830,-47.277,179.686,4.751,148.895
C03207=1116.042,-86.615,-47.286,179.686,4.754,148.896
C03208=1116.038,-86.401,-47.294,179.686,4.758,148.897
C03209=1116.033,-86.184,-47.303,179.685,4.764,148.898
C03210=1116.028,-85.970,-47.311,179.685,4.768,148.899
C03211=1116.024,-85.755,-47.320,179.684,4.772,148.900
C03212=1116.019,-85.505,-47.330,179.684,4.777,148.901
C03213=1116.013,-85.256,-47.340,179.684,4.782,148.903
C03214=1116.007,-85.006,-47.349,179.683,4.787,148.904
C03215=1116.003,-84.756,-47.359,179.683,4.792,148.905
C03216=1115.997,-84.506,-47.370,179.683,4.797,148.906
C03217=1115.992,-84.257,-47.380,179.682,4.802,148.908
C03218=1115.986,-84.007,-47.390,179.682,4.808,148.909
C03219=1115.982,-83.757,-47.400,179.682,4.813,148.910
C03220=1115.976,-83.507,-47.410,179.681,4.817,148.911
C03221=1115.970,-83.257,-47.420,179.681,4.822,148.912
C03222=1115.965,-83.008,-47.430,179.681,4.827,148.913
C03223=1115.961,-82.758,-47.440,179.681,4.833,148.915
C03224=1115.955,-82.508,-47.450,179.680,4.838,148.916
C03225=1115.949,-82.259,-47.460,179.680,4.843,148.917
C03226=1115.944,-82.009,-47.471,179.680,4.848,148.918
C03227=1115.939,-81.759,-47.481,179.679,4.854,148.920
C03228=1115.934,-81.510,-47.491,179.679,4.859,148.921
C03229=1115.929,-81.260,-47.501,179.678,4.863,148.922
C03230=1115.923,-81.010,-47.512,179.678,4.868,148.923
C03231=1115.918,-80.760,-47.522,179.678,4.873,148.924
C03232=1115.912,-80.510,-47.531,179.678,4.878,148.925
C03233=1115.908,-80.260,-47.541,179.678,4.884,148.927
C03234=1115.902,-80.011,-47.551,179.678,4.889,148.928
C03235=1115.896,-79.761,-47.562,179.677,4.894,148.929
C03236=1115.891,-79.511,-47.572,179.677,4.899,148.930
C03237=1115.886,-79.262,-47.582,179.677,4.904,148.931
C03238=1115.880,-79.012,-47.593,179.677,4.909,148.932
C03239=1115.875,-78.762,-47.603,179.677,4.915,148.934
C03240=1115.870,-78.512,-47.613,179.677,4.920,148.935
C03241=1115.865,-78.263,-47.623,179.677,4.925,148.936
C03242=1115.860,-78.013,-47.634,179.676,4.930,148.937
C03243=1115.854,-77.764,-47.645,179.676,4.935,148.938
C03244=1115.849,-77.514,-47.655,179.676,4.940,148.940
C03245=1115.844,-77.264,-47.665,179.676,4.945,148.941
C03246=1115.838,-77.014,-47.676,179.676,4.951,148.942
C03247=1115.833,-76.764,-47.686,179.676,4.957,148.943
C03248=1115.828,-76.515,-47.696,179.676,4.962,148.944
C03249=1115.822,-76.265,-47.707,179.676,4.967,148.945
C03250=1115.817,-76.015,-47.717,179.676,4.972,148.947
C03251=1115.811,-75.765,-47.727,179.676,4.977,148.947
C03252=1115.806,-75.515,-47.738,179.676,4.982,148.949
C03253=1115.802,-75.266,-47.748,179.676,4.987,148.950
C03254=1115.796,-75.017,-47.758,179.676,4.992,148.951
C03255=1115.791,-74.767,-47.769,179.675,4.997,148.952
C03256=1115.786,-74.517,-47.779,179.675,5.002,148.953
C03257=1115.781,-74.267,-47.790,179.676,5.008,148.954
C03258=1115.775,-74.017,-47.800,179.676,5.014,148.956
C03259=1115.770,-73.768,-47.811,179.676,5.018,148.957
C03260=1115.765,-73.553,-47.820,179.675,5.023,148.958
C03261=1115.761,-73.337,-47.829,179.676,5.027,148.959
C03262=1115.756,-73.123,-47.838,179.676,5.032,148.960
C03263=1115.751,-72.907,-47.847,179.676,5.036,148.961
C03264=1115.747,-72.692,-47.856,179.676,5.041,148.961
C03265=1115.743,-72.478,-47.865,179.676,5.045,148.962
C03266=1115.738,-72.263,-47.875,179.676,5.050,148.963
C03267=1115.733,-72.047,-47.884,179.677,5.054,148.964
C03268=1115.728,-71.798,-47.894,179.676,5.060,148.965
C03269=1115.723,-71.548,-47.906,179.676,5.065,148.967
C03270=1115.717,-71.298,-47.916,179.676,5.070,148.968
C03271=1115.712,-71.049,-47.926,179.677,5.075,148.969
C03272=1115.707,-70.799,-47.937,179.677,5.081,148.970
C03273=1115.701,-70.550,-47.947,179.677,5.086,148.971
C03274=1115.696,-70.300,-47.958,179.677,5.090,148.972
C03275=1115.691,-70.050,-47.968,179.677,5.096,148.973
C03276=1115.686,-69.800,-47.979,179.677,5.101,148.974
C03277=1115.681,-69.551,-47.990,179.678,5.106,148.975
C03278=1115.676,-69.301,-48.000,179.678,5.111,148.976
C03279=1115.670,-69.051,-48.012,179.678,5.117,148.977
C03280=1115.665,-68.801,-48.022,179.678,5.121,148.978
C03281=1115.660,-68.551,-48.034,179.679,5.127,148.980
C03282=1115.654,-68.302,-48.044,179.678,5.132,148.981
C03283=1115.649,-68.052,-48.054,179.679,5.137,148.982
C03284=1115.644,-67.803,-48.065,179.679,5.142,148.983
C03285=1115.639,-67.552,-48.076,179.680,5.148,148.984
C03286=1115.634,-67.304,-48.087,179.679,5.153,148.985
C03287=1115.628,-67.053,-48.098,179.680,5.158,148.986
C03288=1115.623,-66.804,-48.109,179.680,5.164,148.987
C03289=1115.618,-66.554,-48.120,179.681,5.169,148.988
C03290=1115.612,-66.304,-48.130,179.681,5.174,148.989
C03291=1115.607,-66.055,-48.141,179.682,5.179,148.990
C03292=1115.602,-65.804,-48.152,179.681,5.184,148.991
C03293=1115.596,-65.555,-48.163,179.682,5.189,148.992
C03294=1115.591,-65.305,-48.174,179.682,5.194,148.993
C03295=1115.586,-65.056,-48.185,179.683,5.200,148.994
C03296=1115.581,-64.806,-48.196,179.683,5.205,148.995
C03297=1115.576,-64.556,-48.207,179.683,5.210,148.996
C03298=1115.570,-64.307,-48.218,179.684,5.215,148.997
C03299=1115.565,-64.057,-48.229,179.684,5.220,148.998
C03300=1115.560,-63.808,-48.240,179.685,5.226,148.999
C03301=1115.554,-63.557,-48.251,179.685,5.231,149.000
C03302=1115.550,-63.308,-48.262,179.686,5.236,149.001
C03303=1115.544,-63.059,-48.273,179.687,5.241,149.002
C03304=1115.539,-62.808,-48.284,179.686,5.246,149.003
C03305=1115.534,-62.558,-48.295,179.687,5.251,149.004
C03306=1115.528,-62.309,-48.306,179.688,5.257,149.005
C03307=1115.524,-62.059,-48.317,179.688,5.261,149.006
C03308=1115.518,-61.809,-48.329,179.688,5.266,149.007
C03309=1115.513,-61.560,-48.339,179.689,5.272,149.008
C03310=1115.508,-61.310,-48.350,179.689,5.277,149.009
C03311=1115.502,-61.060,-48.362,179.690,5.282,149.010
C03312=1115.497,-60.811,-48.372,179.691,5.287,149.011
C03313=1115.492,-60.561,-48.384,179.691,5.292,149.012
C03314=1115.487,-60.311,-48.396,179.692,5.297,149.013
C03315=1115.481,-60.062,-48.406,179.693,5.302,149.013
C03316=1115.477,-59.847,-48.416,179.692,5.306,149.014
C03317=1115.472,-59.632,-48.426,179.692,5.310,149.015
C03318=1115.468,-59.417,-48.436,179.692,5.314,149.016
C03319=1115.463,-59.202,-48.445,179.692,5.319,149.017
C03320=1115.459,-58.987,-48.455,179.692,5.323,149.018
C03321=1115.454,-58.772,-48.465,179.692,5.327,149.019
C03322=1115.450,-58.557,-48.474,179.692,5.331,149.020
C03323=1115.445,-58.342,-48.484,179.692,5.335,149.021
C03324=1115.440,-58.093,-48.495,179.691,5.340,149.022
C03325=1115.436,-57.843,-48.507,179.691,5.344,149.023
C03326=1115.429,-57.593,-48.517,179.691,5.349,149.024
C03327=1115.425,-57.343,-48.529,179.690,5.353,149.025
C03328=1115.419,-57.093,-48.541,179.691,5.358,149.026
C03329=1115.415,-56.844,-48.552,179.691,5.363,149.027
C03330=1115.409,-56.595,-48.563,179.691,5.367,149.028
C03331=1115.404,-56.345,-48.575,179.690,5.372,149.029
C03332=1115.399,-56.095,-48.585,179.690,5.376,149.031
C03333=1115.394,-55.845,-48.597,179.690,5.381,149.031
C03334=1115.388,-55.596,-48.608,179.690,5.386,149.033
C03335=1115.383,-55.346,-48.620,179.689,5.391,149.034
C03336=1115.378,-55.096,-48.631,179.690,5.395,149.035
C03337=1115.373,-54.846,-48.643,179.689,5.400,149.036
C03338=1115.367,-54.597,-48.654,179.689,5.405,149.037
C03339=1115.362,-54.348,-48.666,179.689,5.410,149.038
C03340=1115.357,-54.098,-48.677,179.689,5.414,149.039
C03341=1115.352,-53.847,-48.688,179.689,5.419,149.040
C03342=1115.347,-53.598,-48.700,179.689,5.423,149.041
C03343=1115.341,-53.348,-48.711,179.688,5.428,149.042
C03344=1115.336,-53.099,-48.722,179.688,5.433,149.043
C03345=1115.331,-52.849,-48.734,179.688,5.437,149.044
C03346=1115.326,-52.599,-48.746,179.688,5.442,149.046
C03347=1115.321,-52.349,-48.757,179.688,5.448,149.047
C03348=1115.315,-52.100,-48.768,179.688,5.452,149.048
C03349=1115.310,-51.850,-48.780,179.688,5.457,149.049
C03350=1115.305,-51.601,-48.792,179.687,5.461,149.050
C03351=1115.300,-51.351,-48.803,179.687,5.466,149.051
C03352=1115.295,-51.101,-48.815,179.687,5.471,149.052
C03353=1115.290,-50.851,-48.827,179.687,5.475,149.053
C03354=1115.284,-50.602,-48.838,179.687,5.480,149.054
C03355=1115.279,-50.353,-48.849,179.686,5.484,149.055
C03356=1115.273,-50.103,-48.861,179.686,5.489,149.056
C03357=1115.269,-49.853,-48.873,179.686,5.495,149.057
C03358=1115.263,-49.603,-48.885,179.686,5.498,149.058
C03359=1115.258,-49.353,-48.896,179.686,5.504,149.060
C03360=1115.253,-49.104,-48.907,179.685,5.508,149.061
C03361=1115.247,-48.854,-48.919,179.686,5.513,149.062
C03362=1115.242,-48.605,-48.931,179.686,5.518,149.063
C03363=1115.237,-48.355,-48.943,179.685,5.522,149.064
C03364=1115.232,-48.105,-48.955,179.685,5.527,149.065
C03365=1115.227,-47.856,-48.966,179.685,5.531,149.066
C03366=1115.222,-47.606,-48.978,179.685,5.536,149.067
C03367=1115.216,-47.357,-48.990,179.685,5.542,149.068
C03368=1115.211,-47.107,-49.001,179.684,5.545,149.069
C03369=1115.206,-46.857,-49.013,179.684,5.551,149.070
C03370=1115.201,-46.607,-49.024,179.684,5.556,149.071
C03371=1115.196,-46.357,-49.036,179.684,5.560,149.072
C03372=1115.191,-46.143,-49.047,179.683,5.564,149.074
C03373=1115.187,-45.928,-49.057,179.683,5.568,149.074
C03374=1115.182,-45.713,-49.067,179.683,5.572,149.075
C03375=1115.178,-45.498,-49.077,179.684,5.577,149.076
C03376=1115.173,-45.283,-49.087,179.683,5.581,149.077
C03377=1115.169,-45.069,-49.097,179.683,5.585,149.078
C03378=1115.165,-44.854,-49.107,179.683,5.588,149.079
C03379=1115.160,-44.638,-49.118,179.683,5.592,149.080
C03380=1115.155,-44.389,-49.129,179.683,5.598,149.081
C03381=1115.150,-44.139,-49.141,179.683,5.601,149.082
C03382=1115.144,-43.890,-49.153,179.683,5.607,149.083
C03383=1115.139,-43.641,-49.165,179.682,5.611,149.084
C03384=1115.134,-43.391,-49.177,179.682,5.616,149.085
C03385=1115.128,-43.141,-49.188,179.682,5.621,149.086
C03386=1115.123,-42.891,-49.201,179.682,5.625,149.087
C03387=1115.118,-42.642,-49.212,179.683,5.631,149.088
C03388=1115.113,-42.392,-49.224,179.684,5.636,149.089
C03389=1115.108,-42.142,-49.236,179.685,5.642,149.090
C03390=1115.102,-41.893,-49.249,179.686,5.647,149.091
C03391=1115.098,-41.643,-49.260,179.687,5.652,149.092
C03392=1115.092,-41.393,-49.272,179.688,5.657,149.093
C03393=1115.087,-41.144,-49.284,179.689,5.663,149.094
C03394=1115.082,-40.894,-49.296,179.690,5.667,149.094
C03395=1115.076,-40.644,-49.308,179.691,5.673,149.095
C03396=1115.072,-40.395,-49.320,179.692,5.678,149.096
C03397=1115.067,-40.145,-49.332,179.692,5.683,149.097
C03398=1115.061,-39.895,-49.344,179.694,5.688,149.098
C03399=1115.056,-39.646,-49.357,179.694,5.693,149.099
C03400=1115.051,-39.396,-49.369,179.695,5.698,149.099
C03401=1115.045,-39.146,-49.381,179.696,5.703,149.100
C03402=1115.040,-38.897,-49.393,179.697,5.708,149.101
C03403=1115.036,-38.648,-49.405,179.698,5.713,149.102
C03404=1115.030,-38.398,-49.417,179.698,5.718,149.103
C03405=1115.025,-38.148,-49.429,179.699,5.722,149.104
C03406=1115.020,-37.898,-49.441,179.700,5.727,149.104
C03407=1115.014,-37.648,-49.453,179.701,5.732,149.105
C03408=1115.009,-37.399,-49.466,179.701,5.737,149.106
C03409=1115.004,-37.149,-49.478,179.702,5.742,149.107
C03410=1114.999,-36.900,-49.490,179.702,5.746,149.108
C03411=1114.994,-36.649,-49.503,179.703,5.751,149.109
C03412=1114.989,-36.400,-49.515,179.704,5.755,149.109
C03413=1114.983,-36.151,-49.528,179.704,5.760,149.110
C03414=1114.978,-35.901,-49.540,179.705,5.765,149.111
C03415=1114.973,-35.651,-49.552,179.705,5.770,149.112
C03416=1114.967,-35.401,-49.564,179.706,5.774,149.113
C03417=1114.963,-35.152,-49.576,179.707,5.779,149.114
C03418=1114.958,-34.902,-49.588,179.707,5.783,149.115
C03419=1114.953,-34.653,-49.601,179.707,5.788,149.116
C03420=1114.947,-34.404,-49.613,179.708,5.793,149.116
C03421=1114.943,-34.153,-49.626,179.708,5.796,149.117
C03422=1114.937,-33.904,-49.638,179.709,5.801,149.118
C03423=1114.932,-33.654,-49.650,179.709,5.806,149.119
C03424=1114.927,-33.405,-49.663,179.710,5.811,149.120
C03425=1114.921,-33.155,-49.676,179.709,5.815,149.121
C03426=1114.916,-32.905,-49.688,179.710,5.819,149.122
C03427=1114.910,-32.656,-49.700,179.710,5.824,149.123
C03428=1114.903,-32.260,-49.719,179.710,5.830,149.124
C03429=1114.895,-31.865,-49.740,179.711,5.837,149.125
C03430=1114.886,-31.469,-49.759,179.712,5.845,149.127
C03431=1114.878,-31.073,-49.779,179.711,5.851,149.128
C03432=1114.873,-30.823,-49.792,179.712,5.856,149.129
C03433=1114.868,-30.573,-49.805,179.712,5.860,149.130
C03434=1114.863,-30.324,-49.817,179.712,5.865,149.131
C03435=1114.857,-30.074,-49.829,179.712,5.869,149.132
C03436=1114.852,-29.825,-49.842,179.712,5.873,149.133
C03437=1114.847,-29.575,-49.854,179.712,5.878,149.134
C03438=1114.843,-29.325,-49.867,179.712,5.882,149.135
C03439=1114.838,-29.076,-49.880,179.712,5.886,149.136
C03440=1114.832,-28.826,-49.892,179.712,5.890,149.137
C03441=1114.827,-28.577,-49.904,179.711,5.895,149.138
C03442=1114.821,-28.327,-49.918,179.711,5.899,149.139
C03443=1114.817,-28.077,-49.931,179.712,5.903,149.140
C03444=1114.812,-27.828,-49.943,179.711,5.908,149.141
C03445=1114.806,-27.578,-49.955,179.711,5.912,149.142
C03446=1114.801,-27.329,-49.968,179.710,5.916,149.143
C03447=1114.796,-27.079,-49.981,179.711,5.921,149.144
C03448=1114.791,-26.829,-49.993,179.710,5.925,149.145
C03449=1114.785,-26.580,-50.006,179.710,5.929,149.146
C03450=1114.780,-26.330,-50.019,179.709,5.933,149.147
C03451=1114.775,-26.080,-50.031,179.709,5.938,149.148
C03452=1114.770,-25.830,-50.044,179.709,5.941,149.149
C03453=1114.765,-25.581,-50.057,179.709,5.947,149.150
C03454=1114.760,-25.332,-50.069,179.709,5.951,149.151
C03455=1114.755,-25.081,-50.083,179.710,5.956,149.152
C03456=1114.750,-24.832,-50.095,179.710,5.961,149.153
C03457=1114.745,-24.583,-50.108,179.711,5.966,149.154
C03458=1114.739,-24.333,-50.121,179.712,5.971,149.154
C03459=1114.735,-24.083,-50.133,179.712,5.976,149.155
C03460=1114.729,-23.834,-50.147,179.713,5.981,149.156
C03461=1114.724,-23.584,-50.159,179.713,5.985,149.157
C03462=1114.719,-23.335,-50.171,179.714,5.990,149.158
C03463=1114.714,-23.085,-50.184,179.714,5.995,149.159
C03464=1114.708,-22.835,-50.197,179.715,5.999,149.160
C03465=1114.703,-22.586,-50.210,179.715,6.004,149.161
C03466=1114.699,-22.336,-50.223,179.716,6.009,149.162
C03467=1114.693,-22.086,-50.236,179.716,6.014,149.163
C03468=1114.688,-21.837,-50.249,179.716,6.018,149.163
C03469=1114.682,-21.587,-50.261,179.717,6.023,149.164
C03470=1114.678,-21.337,-50.274,179.718,6.027,149.165
C03471=1114.672,-21.088,-50.288,179.718,6.032,149.166
C03472=1114.667,-20.804,-50.302,179.719,6.038,149.167
C03473=1114.660,-20.521,-50.317,179.720,6.043,149.168
C03474=1114.655,-20.238,-50.331,179.720,6.049,149.169
C03475=1114.649,-19.954,-50.347,179.721,6.053,149.170
C03476=1114.644,-19.705,-50.359,179.721,6.058,149.171
C03477=1114.638,-19.455,-50.372,179.722,6.063,149.172
C03478=1114.634,-19.205,-50.385,179.722,6.068,149.173
C03479=1114.629,-18.956,-50.398,179.723,6.072,149.174
C03480=1114.624,-18.741,-50.409,179.724,6.077,149.174
C03481=1114.620,-18.526,-50.421,179.724,6.080,149.175
C03482=1114.615,-18.311,-50.432,179.724,6.085,149.176
C03483=1114.611,-18.097,-50.443,179.725,6.089,149.176
C03484=1114.607,-17.882,-50.455,179.726,6.093,149.177
C03485=1114.602,-17.667,-50.466,179.726,6.097,149.178
C03486=1114.597,-17.453,-50.477,179.726,6.100,149.179
C03487=1114.593,-17.238,-50.488,179.727,6.105,149.179
C03488=1114.588,-16.989,-50.502,179.727,6.109,149.180
C03489=1114.583,-16.739,-50.515,179.728,6.114,149.181
C03490=1114.578,-16.489,-50.529,179.728,6.119,149.182
C03491=1114.573,-16.240,-50.541,179.729,6.123,149.183
C03492=1114.568,-15.991,-50.554,179.730,6.128,149.184
C03493=1114.563,-15.741,-50.568,179.730,6.133,149.184
C03494=1114.557,-15.491,-50.581,179.731,6.137,149.185
C03495=1114.552,-15.241,-50.594,179.731,6.142,149.186
C03496=1114.547,-14.992,-50.607,179.732,6.146,149.187
C03497=1114.542,-14.742,-50.621,179.733,6.151,149.188
C03498=1114.537,-14.493,-50.634,179.733,6.155,149.189
C03499=1114.532,-14.243,-50.648,179.733,6.160,149.190
C03500=1114.527,-13.994,-50.661,179.734,6.164,149.190
C03501=1114.521,-13.744,-50.674,179.735,6.169,149.191
C03502=1114.517,-13.494,-50.687,179.735,6.174,149.192
C03503=1114.511,-13.245,-50.701,179.736,6.178,149.193
C03504=1114.506,-12.995,-50.714,179.736,6.183,149.194
C03505=1114.501,-12.746,-50.727,179.737,6.187,149.195
C03506=1114.496,-12.496,-50.740,179.738,6.192,149.195
C03507=1114.491,-12.246,-50.754,179.738,6.197,149.196
C03508=1114.486,-11.997,-50.767,179.739,6.202,149.197
C03509=1114.480,-11.747,-50.781,179.740,6.206,149.198
C03510=1114.476,-11.498,-50.794,179.740,6.211,149.199
C03511=1114.470,-11.248,-50.807,179.741,6.215,149.200
C03512=1114.465,-10.998,-50.821,179.742,6.220,149.200
C03513=1114.460,-10.749,-50.834,179.742,6.224,149.201
C03514=1114.455,-10.499,-50.848,179.742,6.228,149.202
C03515=1114.450,-10.250,-50.861,179.743,6.233,149.203
C03516=1114.445,-10.000,-50.875,179.744,6.237,149.204
C03517=1114.440,-9.750,-50.889,179.744,6.242,149.205
C03518=1114.435,-9.501,-50.902,179.745,6.247,149.205
C03519=1114.430,-9.251,-50.916,179.745,6.252,149.206
C03520=1114.425,-9.002,-50.928,179.746,6.256,149.207
C03521=1114.420,-8.752,-50.943,179.747,6.261,149.208
C03522=1114.414,-8.503,-50.956,179.747,6.265,149.209
C03523=1114.410,-8.253,-50.970,179.748,6.270,149.209
C03524=1114.404,-8.004,-50.983,179.749,6.274,149.210
C03525=1114.399,-7.754,-50.997,179.748,6.278,149.211
C03526=1114.394,-7.504,-51.010,179.749,6.283,149.212
C03527=1114.389,-7.255,-51.024,179.750,6.287,149.213
C03528=1114.384,-7.005,-51.038,179.750,6.292,149.214
C03529=1114.379,-6.756,-51.051,179.751,6.297,149.215
C03530=1114.374,-6.506,-51.065,179.752,6.301,149.215
C03531=1114.368,-6.256,-51.078,179.753,6.306,149.216
C03532=1114.364,-6.007,-51.092,179.753,6.311,149.217
C03533=1114.359,-5.757,-51.106,179.754,6.315,149.218
C03534=1114.353,-5.508,-51.119,179.755,6.320,149.219
C03535=1114.348,-5.258,-51.134,179.754,6.324,149.219
C03536=1114.343,-5.043,-51.145,179.755,6.328,149.220
C03537=1114.339,-4.829,-51.157,179.756,6.332,149.221
C03538=1114.335,-4.614,-51.169,179.757,6.336,149.221
C03539=1114.331,-4.400,-51.181,179.757,6.340,149.222
C03540=1114.326,-4.185,-51.193,179.757,6.343,149.223
C03541=1114.322,-3.970,-51.205,179.758,6.348,149.224
C03542=1114.317,-3.756,-51.216,179.759,6.351,149.224
C03543=1114.313,-3.541,-51.229,179.759,6.355,149.225
C03544=1114.308,-3.292,-51.242,179.759,6.359,149.226
C03545=1114.303,-3.042,-51.255,179.760,6.364,149.227
C03546=1114.298,-2.793,-51.269,179.761,6.369,149.227
C03547=1114.293,-2.543,-51.284,179.761,6.373,149.228
C03548=1114.288,-2.293,-51.297,179.762,6.378,149.229
C03549=1114.282,-2.044,-51.311,179.763,6.383,149.230
C03550=1114.278,-1.795,-51.325,179.764,6.387,149.231
C03551=1114.273,-1.545,-51.339,179.763,6.391,149.232
C03552=1114.267,-1.296,-51.353,179.764,6.396,149.233
C03553=1114.262,-1.046,-51.367,179.765,6.400,149.233
C03554=1114.257,-0.796,-51.381,179.765,6.405,149.234
C03555=1114.252,-0.546,-51.395,179.766,6.409,149.235
C03556=1114.247,-0.298,-51.408,179.767,6.414,149.236
C03557=1114.242,-0.048,-51.423,179.768,6.418,149.237
C03558=1114.237,0.202,-51.437,179.768,6.423,149.237
C03559=1114.232,0.451,-51.450,179.769,6.428,149.238
C03560=1114.227,0.701,-51.464,179.769,6.432,149.239
C03561=1114.222,0.951,-51.479,179.770,6.436,149.240
C03562=1114.217,1.201,-51.493,179.770,6.441,149.241
C03563=1114.211,1.450,-51.507,179.771,6.446,149.242
C03564=1114.206,1.699,-51.521,179.771,6.450,149.243
C03565=1114.202,1.949,-51.535,179.772,6.455,149.243
C03566=1114.197,2.198,-51.549,179.773,6.459,149.244
C03567=1114.191,2.447,-51.563,179.773,6.464,149.245
C03568=1114.187,2.697,-51.577,179.774,6.469,149.246
C03569=1114.182,2.947,-51.592,179.774,6.472,149.247
C03570=1114.177,3.197,-51.606,179.775,6.477,149.247
C03571=1114.171,3.446,-51.620,179.775,6.482,149.248
C03572=1114.166,3.695,-51.634,179.776,6.486,149.249
C03573=1114.161,3.945,-51.648,179.777,6.491,149.250
C03574=1114.156,4.195,-51.663,179.777,6.495,149.251
C03575=1114.151,4.444,-51.677,179.778,6.500,149.252
C03576=1114.146,4.693,-51.691,179.778,6.505,149.253
C03577=1114.141,4.943,-51.705,179.779,6.509,149.253
C03578=1114.136,5.193,-51.719,179.780,6.514,149.254
C03579=1114.131,5.443,-51.734,179.780,6.518,149.255
C03580=1114.125,5.692,-51.748,179.780,6.523,149.256
C03581=1114.120,5.941,-51.762,179.781,6.527,149.257
C03582=1114.115,6.191,-51.776,179.781,6.532,149.258
C03583=1114.110,6.441,-51.790,179.782,6.536,149.258
C03584=1114.105,6.690,-51.805,179.783,6.541,149.259
C03585=1114.100,6.940,-51.819,179.784,6.546,149.260
C03586=1114.095,7.189,-51.833,179.784,6.550,149.261
C03587=1114.090,7.439,-51.847,179.785,6.555,149.262
C03588=1114.085,7.688,-51.862,179.785,6.560,149.263
C03589=1114.080,7.938,-51.876,179.786,6.564,149.263
C03590=1114.075,8.187,-51.891,179.787,6.569,149.264
C03591=1114.070,8.437,-51.906,179.787,6.573,149.265
C03592=1114.065,8.651,-51.918,179.788,6.577,149.266
C03593=1114.061,8.866,-51.930,179.788,6.581,149.267
C03594=1114.056,9.080,-51.943,179.789,6.585,149.267
C03595=1114.052,9.295,-51.955,179.789,6.589,149.268
C03596=1114.048,9.509,-51.967,179.789,6.593,149.269
C03597=1114.044,9.723,-51.979,179.790,6.597,149.270
C03598=1114.039,9.938,-51.992,179.790,6.601,149.270
C03599=1114.036,10.153,-52.005,179.791,6.604,149.271
C03600=1114.030,10.402,-52.019,179.791,6.609,149.272
C03601=1114.025,10.652,-52.033,179.792,6.614,149.273
C03602=1114.019,10.902,-52.048,179.793,6.618,149.274
C03603=1114.015,11.151,-52.063,179.793,6.623,149.274
C03604=1114.010,11.401,-52.077,179.794,6.627,149.275
C03605=1114.005,11.650,-52.091,179.795,6.632,149.276
C03606=1114.000,11.899,-52.106,179.795,6.637,149.277
C03607=1113.995,12.149,-52.121,179.796,6.642,149.278
C03608=1113.989,12.399,-52.136,179.797,6.646,149.278
C03609=1113.985,12.648,-52.151,179.797,6.650,149.279
C03610=1113.980,12.898,-52.165,179.797,6.655,149.280
C03611=1113.975,13.148,-52.179,179.798,6.659,149.281
C03612=1113.970,13.397,-52.195,179.799,6.664,149.282
C03613=1113.964,13.646,-52.209,179.799,6.668,149.283
C03614=1113.959,13.896,-52.223,179.800,6.673,149.283
C03615=1113.954,14.145,-52.238,179.801,6.677,149.284
C03616=1113.949,14.395,-52.252,179.802,6.682,149.285
C03617=1113.944,14.644,-52.268,179.803,6.686,149.286
C03618=1113.939,14.894,-52.282,179.803,6.690,149.287
C03619=1113.934,15.143,-52.296,179.803,6.695,149.287
C03620=1113.929,15.393,-52.312,179.804,6.699,149.288
C03621=1113.924,15.642,-52.326,179.805,6.704,149.289
C03622=1113.919,15.892,-52.341,179.806,6.708,149.290
C03623=1113.914,16.141,-52.355,179.806,6.713,149.290
C03624=1113.909,16.391,-52.371,179.807,6.718,149.291
C03625=1113.904,16.640,-52.385,179.808,6.722,149.292
C03626=1113.899,16.889,-52.400,179.808,6.726,149.293
C03627=1113.893,17.139,-52.415,179.809,6.730,149.294
C03628=1113.889,17.389,-52.430,179.809,6.735,149.294
C03629=1113.884,17.638,-52.444,179.810,6.739,149.295
C03630=1113.879,17.888,-52.460,179.811,6.744,149.296
C03631=1113.874,18.137,-52.474,179.812,6.748,149.297
C03632=1113.869,18.386,-52.489,179.813,6.753,149.297
C03633=1113.863,18.637,-52.504,179.814,6.757,149.298
C03634=1113.859,18.886,-52.519,179.814,6.761,149.299
C03635=1113.854,19.135,-52.533,179.815,6.766,149.300
C03636=1113.849,19.385,-52.549,179.815,6.770,149.301
C03637=1113.844,19.635,-52.564,179.816,6.775,149.301
C03638=1113.838,19.885,-52.579,179.817,6.779,149.302
C03639=1113.834,20.134,-52.594,179.818,6.784,149.303
C03640=1113.829,20.383,-52.609,179.818,6.788,149.304
C03641=1113.823,20.633,-52.624,179.819,6.793,149.304
C03642=1113.819,20.882,-52.639,179.819,6.797,149.305
C03643=1113.813,21.132,-52.654,179.820,6.801,149.306
C03644=1113.808,21.381,-52.669,179.822,6.805,149.306
C03645=1113.803,21.630,-52.685,179.822,6.810,149.307
C03646=1113.798,21.880,-52.699,179.823,6.814,149.308
C03647=1113.794,22.129,-52.714,179.824,6.818,149.309
C03648=1113.789,22.344,-52.727,179.825,6.822,149.309
C03649=1113.785,22.558,-52.741,179.825,6.826,149.310
C03650=1113.781,22.773,-52.753,179.826,6.830,149.311
C03651=1113.776,22.987,-52.767,179.827,6.833,149.311
